LIN {X 0,Y 386.011,Z 375.259,A -85,B 0,C 180,E1 14858.04,E2 14858.04} C_VEL
LIN {X 0,Y 386.531,Z 375.685,A -85,B 0,C 180,E1 14854.451,E2 14854.451} C_VEL
LIN {X 0,Y 386.714,Z 375.838,A -85,B 0,C 180,E1 14850.889,E2 14850.889} C_VEL
LIN {X 0,Y 386.655,Z 375.781,A -85,B 0,C 180,E1 14847.184,E2 14847.184} C_VEL
LIN {X 0,Y 386.291,Z 375.479,A -85,B 0,C 180,E1 14843.61,E2 14843.61} C_VEL
LIN {X 0,Y 385.591,Z 374.785,A -85,B 0,C 180,E1 14839.693,E2 14839.693} C_VEL
LIN {X 0,Y 384.724,Z 373.685,A -85,B 0,C 180,E1 14836.167,E2 14836.167} C_VEL
LIN {X 0,Y 383.625,Z 371.619,A -85,B 0,C 180,E1 14832.559,E2 14832.559} C_VEL
LIN {X 0,Y 382.556,Z 370.431,A -85,B 0,C 180,E1 14829.766,E2 14829.766} C_VEL
LIN {X 0,Y 380.821,Z 369.656,A -85,B 0,C 180,E1 14826.151,E2 14826.151} C_VEL
LIN {X 0,Y 378.919,Z 368.36,A -85,B 0,C 180,E1 14822.669,E2 14822.669} C_VEL
LIN {X 0,Y 377.138,Z 366.192,A -85,B 0,C 180,E1 14819.5,E2 14819.5} C_VEL
LIN {X 0,Y 375.495,Z 363.505,A -85,B 0,C 180,E1 14816.731,E2 14816.731} C_VEL
LIN {X 0,Y 372.832,Z 362.159,A -85,B 0,C 180,E1 14813.051,E2 14813.051} C_VEL
LIN {X 0,Y 370.445,Z 359.93,A -85,B 0,C 180,E1 14809.83,E2 14809.83} C_VEL
LIN {X 0,Y 368.756,Z 357.1,A -85,B 0,C 180,E1 14807.52,E2 14807.52} C_VEL
LIN {X 0,Y 367.813,Z 356.251,A -85,B 0,C 180,E1 14806.31,E2 14806.31} C_VEL
LIN {X 0,Y 364.925,Z 354.532,A -85,B 0,C 180,E1 14802.985,E2 14802.985} C_VEL
LIN {X 0,Y 362.696,Z 352.012,A -85,B 0,C 180,E1 14800.378,E2 14800.378} C_VEL
LIN {X 0,Y 361.179,Z 349.438,A -85,B 0,C 180,E1 14798.526,E2 14798.526} C_VEL
LIN {X 0,Y 358.071,Z 347.716,A -85,B 0,C 180,E1 14795.311,E2 14795.311} C_VEL
LIN {X 0,Y 355.633,Z 344.996,A -85,B 0,C 180,E1 14792.67,E2 14792.67} C_VEL
LIN {X 0,Y 354.249,Z 342.492,A -85,B 0,C 180,E1 14791.099,E2 14791.099} C_VEL
LIN {X 0,Y 350.886,Z 340.633,A -85,B 0,C 180,E1 14787.86,E2 14787.86} C_VEL
LIN {X 0,Y 348.108,Z 337.648,A -85,B 0,C 180,E1 14785.43,E2 14785.43} C_VEL
LIN {X 0,Y 346.58,Z 335.327,A -85,B 0,C 180,E1 14784.183,E2 14784.183} C_VEL
LIN {X 0,Y 344.787,Z 334.431,A -85,B 0,C 180,E1 14782.943,E2 14782.943} C_VEL
LIN {X 0,Y 343.15,Z 334.686,A -85,B 0,C 180,E1 14781.962,E2 14781.962} C_VEL
LIN {X 0,Y 339.462,Z 337.058,A -85,B 0,C 180,E1 14780.04,E2 14780.04} C_VEL
LIN {X 0,Y 337.971,Z 336.456,A -85,B 0,C 180,E1 14779.212,E2 14779.212} C_VEL
LIN {X 0,Y 337.791,Z 336.192,A -85,B 0,C 180,E1 14779.1,E2 14779.1} C_VEL
LIN {X 0,Y 333.793,Z 333.025,A -85,B 0,C 180,E1 14776.712,E2 14776.712} C_VEL
LIN {X 0,Y 331.304,Z 329.103,A -85,B 0,C 180,E1 14774.864,E2 14774.864} C_VEL
LIN {X 0,Y 327.846,Z 326.408,A -85,B 0,C 180,E1 14772.058,E2 14772.058} C_VEL
LIN {X 0,Y 325.939,Z 322.868,A -85,B 0,C 180,E1 14769.892,E2 14769.892} C_VEL
LIN {X 0,Y 321.747,Z 319.853,A -85,B 0,C 180,E1 14761.425,E2 14761.425} C_VEL
LIN {X 0,Y 322.04,Z 320.213,A -85,B 0,C 180,E1 14757.331,E2 14757.331} C_VEL
LIN {X 0,Y 326.157,Z 323.109,A -85,B 0,C 180,E1 14750.293,E2 14750.293} C_VEL
LIN {X 0,Y 327.926,Z 326.507,A -85,B 0,C 180,E1 14748.302,E2 14748.302} C_VEL
LIN {X 0,Y 331.172,Z 329.042,A -85,B 0,C 180,E1 14745.666,E2 14745.666} C_VEL
LIN {X 0,Y 331.836,Z 329.903,A -85,B 0,C 180,E1 14745.16,E2 14745.16} C_VEL
LIN {X 0,Y 334.411,Z 333.737,A -85,B 0,C 180,E1 14743.32,E2 14743.32} C_VEL
LIN {X 0,Y 336.959,Z 335.929,A -85,B 0,C 180,E1 14741.802,E2 14741.802} C_VEL
LIN {X 0,Y 340.182,Z 340.253,A -85,B 0,C 180,E1 14739.976,E2 14739.976} C_VEL
LIN {X 0,Y 341.916,Z 342.055,A -85,B 0,C 180,E1 14739.099,E2 14739.099} C_VEL
LIN {X 0,Y 345.521,Z 346.558,A -85,B 0,C 180,E1 14737.364,E2 14737.364} C_VEL
LIN {X 0,Y 351.232,Z 353.852,A -85,B 0,C 180,E1 14734.903,E2 14734.903} C_VEL
LIN {X 0,Y 355.157,Z 359.117,A -85,B 0,C 180,E1 14733.364,E2 14733.364} C_VEL
LIN {X 0,Y 362.926,Z 371.553,A -85,B 0,C 180,E1 14730.543,E2 14730.543} C_VEL
LIN {X 0,Y 370.435,Z 384.324,A -85,B 0,C 180,E1 14728.106,E2 14728.106} C_VEL
LIN {X 0,Y 378.916,Z 400.148,A -85,B 0,C 180,E1 14725.596,E2 14725.596} C_VEL
LIN {X 0,Y 379.902,Z 402.489,A -85,B 0,C 180,E1 14725.306,E2 14725.306} C_VEL
LIN {X 0,Y 368.607,Z 600.449,A -85,B 0,C 180,E1 14721.342,E2 14721.342} C_VEL
LIN {X 0,Y 366.108,Z 623.413,A -85,B 0,C 180,E1 14720.702,E2 14720.702} C_VEL
LIN {X 0,Y 363.074,Z 642.585,A -85,B 0,C 180,E1 14719.956,E2 14719.956} C_VEL
LIN {X 0,Y 359.795,Z 659.806,A -85,B 0,C 180,E1 14719.1,E2 14719.1} C_VEL
LIN {X 0,Y 355.353,Z 679.953,A -85,B 0,C 180,E1 14717.85,E2 14717.85} C_VEL
LIN {X 0,Y 350.278,Z 699.216,A -85,B 0,C 180,E1 14716.34,E2 14716.34} C_VEL
LIN {X 0,Y 345.77,Z 714.793,A -85,B 0,C 180,E1 14714.874,E2 14714.874} C_VEL
LIN {X 0,Y 340.805,Z 730.632,A -85,B 0,C 180,E1 14713.122,E2 14713.122} C_VEL
LIN {X 0,Y 334.365,Z 749.665,A -85,B 0,C 180,E1 14710.576,E2 14710.576} C_VEL
LIN {X 0,Y 329.444,Z 763.462,A -85,B 0,C 180,E1 14708.363,E2 14708.363} C_VEL
LIN {X 0,Y 324.527,Z 776.993,A -85,B 0,C 180,E1 14705.829,E2 14705.829} C_VEL
LIN {X 0,Y 318.929,Z 792.167,A -85,B 0,C 180,E1 14702.417,E2 14702.417} C_VEL
LIN {X 0,Y 314.992,Z 803.107,A -85,B 0,C 180,E1 14699.472,E2 14699.472} C_VEL
LIN {X 0,Y 311.188,Z 814.397,A -85,B 0,C 180,E1 14695.888,E2 14695.888} C_VEL
LIN {X 0,Y 308.203,Z 824.017,A -85,B 0,C 180,E1 14692.105,E2 14692.105} C_VEL
LIN {X 0,Y 306.371,Z 830.914,A -85,B 0,C 180,E1 14688.839,E2 14688.839} C_VEL
LIN {X 0,Y 305.04,Z 837.21,A -85,B 0,C 180,E1 14685.202,E2 14685.202} C_VEL
LIN {X 0,Y 304.236,Z 842.687,A -85,B 0,C 180,E1 14680.988,E2 14680.988} C_VEL
LIN {X 0,Y 303.996,Z 845.821,A -85,B 0,C 180,E1 14677.56,E2 14677.56} C_VEL
LIN {X 0,Y 303.952,Z 847.721,A -85,B 0,C 180,E1 14674.339,E2 14674.339} C_VEL
LIN {X 0,Y 303.961,Z 848.599,A -85,B 0,C 180,E1 14671.131,E2 14671.131} C_VEL
LIN {X 0,Y 303.955,Z 848.433,A -85,B 0,C 180,E1 14667.738,E2 14667.738} C_VEL
LIN {X 0,Y 303.963,Z 846.79,A -85,B 0,C 180,E1 14663.768,E2 14663.768} C_VEL
LIN {X 0,Y 304.125,Z 843.858,A -85,B 0,C 180,E1 14660.157,E2 14660.157} C_VEL
LIN {X 0,Y 304.586,Z 839.894,A -85,B 0,C 180,E1 14656.716,E2 14656.716} C_VEL
LIN {X 0,Y 305.586,Z 834.412,A -85,B 0,C 180,E1 14653.071,E2 14653.071} C_VEL
LIN {X 0,Y 307.593,Z 826.186,A -85,B 0,C 180,E1 14648.85,E2 14648.85} C_VEL
LIN {X 0,Y 309.881,Z 818.374,A -85,B 0,C 180,E1 14645.607,E2 14645.607} C_VEL
LIN {X 0,Y 312.881,Z 809.224,A -85,B 0,C 180,E1 14642.396,E2 14642.396} C_VEL
LIN {X 0,Y 317.628,Z 795.763,A -85,B 0,C 180,E1 14638.498,E2 14638.498} C_VEL
LIN {X 0,Y 321.804,Z 784.311,A -85,B 0,C 180,E1 14635.738,E2 14635.738} C_VEL
LIN {X 0,Y 326.663,Z 771.157,A -85,B 0,C 180,E1 14633.023,E2 14633.023} C_VEL
LIN {X 0,Y 332.804,Z 754.126,A -85,B 0,C 180,E1 14630.103,E2 14630.103} C_VEL
LIN {X 0,Y 337.815,Z 739.613,A -85,B 0,C 180,E1 14628.018,E2 14628.018} C_VEL
LIN {X 0,Y 343.135,Z 723.386,A -85,B 0,C 180,E1 14626.032,E2 14626.032} C_VEL
LIN {X 0,Y 348.815,Z 704.431,A -85,B 0,C 180,E1 14624.12,E2 14624.12} C_VEL
LIN {X 0,Y 353.278,Z 687.915,A -85,B 0,C 180,E1 14622.741,E2 14622.741} C_VEL
LIN {X 0,Y 357.676,Z 669.757,A -85,B 0,C 180,E1 14621.483,E2 14621.483} C_VEL
LIN {X 0,Y 362.253,Z 647.281,A -85,B 0,C 180,E1 14620.257,E2 14620.257} C_VEL
LIN {X 0,Y 365.247,Z 629.114,A -85,B 0,C 180,E1 14619.502,E2 14619.502} C_VEL
LIN {X 0,Y 367.731,Z 609.909,A -85,B 0,C 180,E1 14618.895,E2 14618.895} C_VEL
LIN {X 0,Y 369.86,Z 580.866,A -85,B 0,C 180,E1 14618.239,E2 14618.239} C_VEL
LIN {X 0,Y 379.865,Z 402.063,A -85,B 0,C 180,E1 14614.672,E2 14614.672} C_VEL
LIN {X 0,Y 372.117,Z 387.455,A -85,B 0,C 180,E1 14612.415,E2 14612.415} C_VEL
LIN {X 0,Y 365.916,Z 376.518,A -85,B 0,C 180,E1 14610.456,E2 14610.456} C_VEL
LIN {X 0,Y 360.022,Z 366.838,A -85,B 0,C 180,E1 14608.443,E2 14608.443} C_VEL
LIN {X 0,Y 353.711,Z 357.015,A -85,B 0,C 180,E1 14606.076,E2 14606.076} C_VEL
LIN {X 0,Y 349.294,Z 351.398,A -85,B 0,C 180,E1 14604.298,E2 14604.298} C_VEL
LIN {X 0,Y 345.346,Z 346.397,A -85,B 0,C 180,E1 14602.558,E2 14602.558} C_VEL
LIN {X 0,Y 341.766,Z 341.796,A -85,B 0,C 180,E1 14600.821,E2 14600.821} C_VEL
LIN {X 0,Y 337.557,Z 336.961,A -85,B 0,C 180,E1 14598.567,E2 14598.567} C_VEL
LIN {X 0,Y 336.628,Z 335.401,A -85,B 0,C 180,E1 14597.993,E2 14597.993} C_VEL
LIN {X 0,Y 333.408,Z 332.568,A -85,B 0,C 180,E1 14596.016,E2 14596.016} C_VEL
LIN {X 0,Y 331.41,Z 329.161,A -85,B 0,C 180,E1 14594.502,E2 14594.502} C_VEL
LIN {X 0,Y 327.926,Z 326.505,A -85,B 0,C 180,E1 14591.698,E2 14591.698} C_VEL
LIN {X 0,Y 326.003,Z 322.973,A -85,B 0,C 180,E1 14589.533,E2 14589.533} C_VEL
LIN {X 0,Y 321.774,Z 319.91,A -85,B 0,C 180,E1 14581.246,E2 14581.246} C_VEL
LIN {X 0,Y 321.978,Z 320.151,A -85,B 0,C 180,E1 14577.152,E2 14577.152} C_VEL
LIN {X 0,Y 326.163,Z 323.134,A -85,B 0,C 180,E1 14569.848,E2 14569.848} C_VEL
LIN {X 0,Y 328.026,Z 326.626,A -85,B 0,C 180,E1 14567.77,E2 14567.77} C_VEL
LIN {X 0,Y 331.694,Z 329.582,A -85,B 0,C 180,E1 14564.841,E2 14564.841} C_VEL
LIN {X 0,Y 334.299,Z 333.596,A -85,B 0,C 180,E1 14562.956,E2 14562.956} C_VEL
LIN {X 0,Y 337.907,Z 336.386,A -85,B 0,C 180,E1 14560.826,E2 14560.826} C_VEL
LIN {X 0,Y 340.872,Z 340.262,A -85,B 0,C 180,E1 14558.942,E2 14558.942} C_VEL
LIN {X 0,Y 344.246,Z 342.664,A -85,B 0,C 180,E1 14556.733,E2 14556.733} C_VEL
LIN {X 0,Y 345.62,Z 343.626,A -85,B 0,C 180,E1 14555.745,E2 14555.745} C_VEL
LIN {X 0,Y 347.956,Z 346.835,A -85,B 0,C 180,E1 14553.827,E2 14553.827} C_VEL
LIN {X 0,Y 350.713,Z 349.153,A -85,B 0,C 180,E1 14551.383,E2 14551.383} C_VEL
LIN {X 0,Y 353.32,Z 350.716,A -85,B 0,C 180,E1 14548.811,E2 14548.811} C_VEL
LIN {X 0,Y 355.344,Z 354.06,A -85,B 0,C 180,E1 14546.53,E2 14546.53} C_VEL
LIN {X 0,Y 358.406,Z 356.549,A -85,B 0,C 180,E1 14543.345,E2 14543.345} C_VEL
LIN {X 0,Y 360.372,Z 357.729,A -85,B 0,C 180,E1 14541.27,E2 14541.27} C_VEL
LIN {X 0,Y 362.586,Z 361.266,A -85,B 0,C 180,E1 14538.562,E2 14538.562} C_VEL
LIN {X 0,Y 365.41,Z 363.514,A -85,B 0,C 180,E1 14535.314,E2 14535.314} C_VEL
LIN {X 0,Y 367.493,Z 364.663,A -85,B 0,C 180,E1 14532.857,E2 14532.857} C_VEL
LIN {X 0,Y 369.237,Z 367.669,A -85,B 0,C 180,E1 14530.455,E2 14530.455} C_VEL
LIN {X 0,Y 371.484,Z 369.86,A -85,B 0,C 180,E1 14527.439,E2 14527.439} C_VEL
LIN {X 0,Y 374.035,Z 371.221,A -85,B 0,C 180,E1 14523.964,E2 14523.964} C_VEL
LIN {X 0,Y 375.036,Z 372.228,A -85,B 0,C 180,E1 14522.402,E2 14522.402} C_VEL
LIN {X 0,Y 376.884,Z 375.227,A -85,B 0,C 180,E1 14519.212,E2 14519.212} C_VEL
LIN {X 0,Y 378.863,Z 377.028,A -85,B 0,C 180,E1 14515.645,E2 14515.645} C_VEL
LIN {X 0,Y 380.652,Z 377.988,A -85,B 0,C 180,E1 14512.224,E2 14512.224} C_VEL
LIN {X 0,Y 382.225,Z 378.874,A -85,B 0,C 180,E1 14508.747,E2 14508.747} C_VEL
LIN {X 0,Y 383.348,Z 380.95,A -85,B 0,C 180,E1 14505.195,E2 14505.195} C_VEL
LIN {X 0,Y 384.312,Z 382.396,A -85,B 0,C 180,E1 14501.708,E2 14501.708} C_VEL
LIN {X 0,Y 385.001,Z 383.161,A -85,B 0,C 180,E1 14498.212,E2 14498.212} C_VEL
LIN {X 0,Y 385.54,Z 383.608,A -85,B 0,C 180,E1 14494.611,E2 14494.611} C_VEL
LIN {X 0,Y 385.734,Z 383.773,A -85,B 0,C 180,E1 14491.04,E2 14491.04} C_VEL
LIN {X 0,Y 385.691,Z 383.733,A -85,B 0,C 180,E1 14487.326,E2 14487.326} C_VEL
LIN {X 0,Y 385.333,Z 383.446,A -85,B 0,C 180,E1 14483.744,E2 14483.744} C_VEL
LIN {X 0,Y 384.675,Z 382.815,A -85,B 0,C 180,E1 14479.971,E2 14479.971} C_VEL
LIN {X 0,Y 383.829,Z 381.752,A -85,B 0,C 180,E1 14476.441,E2 14476.441} C_VEL
LIN {X 0,Y 382.796,Z 379.785,A -85,B 0,C 180,E1 14472.937,E2 14472.937} C_VEL
LIN {X 0,Y 381.65,Z 378.409,A -85,B 0,C 180,E1 14469.929,E2 14469.929} C_VEL
LIN {X 0,Y 379.891,Z 377.628,A -85,B 0,C 180,E1 14466.254,E2 14466.254} C_VEL
LIN {X 0,Y 377.969,Z 376.351,A -85,B 0,C 180,E1 14462.727,E2 14462.727} C_VEL
LIN {X 0,Y 376.128,Z 374.16,A -85,B 0,C 180,E1 14459.461,E2 14459.461} C_VEL
LIN {X 0,Y 374.453,Z 371.411,A -85,B 0,C 180,E1 14456.63,E2 14456.63} C_VEL
LIN {X 0,Y 371.78,Z 370.066,A -85,B 0,C 180,E1 14452.958,E2 14452.958} C_VEL
LIN {X 0,Y 369.397,Z 367.862,A -85,B 0,C 180,E1 14449.756,E2 14449.756} C_VEL
LIN {X 0,Y 367.651,Z 365.01,A -85,B 0,C 180,E1 14447.378,E2 14447.378} C_VEL
LIN {X 0,Y 366.773,Z 364.175,A -85,B 0,C 180,E1 14446.254,E2 14446.254} C_VEL
LIN {X 0,Y 363.902,Z 362.485,A -85,B 0,C 180,E1 14442.953,E2 14442.953} C_VEL
LIN {X 0,Y 361.585,Z 359.928,A -85,B 0,C 180,E1 14440.255,E2 14440.255} C_VEL
LIN {X 0,Y 359.927,Z 357.29,A -85,B 0,C 180,E1 14438.278,E2 14438.278} C_VEL
LIN {X 0,Y 356.842,Z 355.495,A -85,B 0,C 180,E1 14435.058,E2 14435.058} C_VEL
LIN {X 0,Y 354.391,Z 352.74,A -85,B 0,C 180,E1 14432.415,E2 14432.415} C_VEL
LIN {X 0,Y 353.016,Z 350.332,A -85,B 0,C 180,E1 14430.841,E2 14430.841} C_VEL
LIN {X 0,Y 349.525,Z 348.336,A -85,B 0,C 180,E1 14427.53,E2 14427.53} C_VEL
LIN {X 0,Y 346.676,Z 345.239,A -85,B 0,C 180,E1 14425.085,E2 14425.085} C_VEL
LIN {X 0,Y 345.201,Z 343.121,A -85,B 0,C 180,E1 14423.923,E2 14423.923} C_VEL
LIN {X 0,Y 341.517,Z 340.835,A -85,B 0,C 180,E1 14421.467,E2 14421.467} C_VEL
LIN {X 0,Y 338.685,Z 337.568,A -85,B 0,C 180,E1 14419.658,E2 14419.658} C_VEL
LIN {X 0,Y 337.791,Z 336.192,A -85,B 0,C 180,E1 14419.1,E2 14419.1} C_VEL
LIN {X 0,Y 336.204,Z 334.673,A -85,B 0,C 180,E1 14418.145,E2 14418.145} C_VEL
LIN {X 0,Y 333.608,Z 334.681,A -85,B 0,C 180,E1 14416.692,E2 14416.692} C_VEL
LIN {X 0,Y 329.248,Z 336.176,A -85,B 0,C 180,E1 14414.065,E2 14414.065} C_VEL
LIN {X 0,Y 328.115,Z 335.75,A -85,B 0,C 180,E1 14413.204,E2 14413.204} C_VEL
LIN {X 0,Y 325.562,Z 332.515,A -85,B 0,C 180,E1 14410.708,E2 14410.708} C_VEL
LIN {X 0,Y 324.672,Z 330.612,A -85,B 0,C 180,E1 14409.573,E2 14409.573} C_VEL
LIN {X 0,Y 320.755,Z 327.77,A -85,B 0,C 180,E1 14401.25,E2 14401.25} C_VEL
LIN {X 0,Y 321.109,Z 328.228,A -85,B 0,C 180,E1 14397.144,E2 14397.144} C_VEL
LIN {X 0,Y 324.884,Z 330.824,A -85,B 0,C 180,E1 14390.612,E2 14390.612} C_VEL
LIN {X 0,Y 326.681,Z 334.309,A -85,B 0,C 180,E1 14388.525,E2 14388.525} C_VEL
LIN {X 0,Y 330.243,Z 337.376,A -85,B 0,C 180,E1 14385.58,E2 14385.58} C_VEL
LIN {X 0,Y 332.929,Z 341.425,A -85,B 0,C 180,E1 14383.602,E2 14383.602} C_VEL
LIN {X 0,Y 335.288,Z 343.541,A -85,B 0,C 180,E1 14382.157,E2 14382.157} C_VEL
LIN {X 0,Y 338.76,Z 348.09,A -85,B 0,C 180,E1 14380.158,E2 14380.158} C_VEL
LIN {X 0,Y 340.22,Z 349.818,A -85,B 0,C 180,E1 14379.395,E2 14379.395} C_VEL
LIN {X 0,Y 344.789,Z 355.602,A -85,B 0,C 180,E1 14377.178,E2 14377.178} C_VEL
LIN {X 0,Y 349.224,Z 361.396,A -85,B 0,C 180,E1 14375.246,E2 14375.246} C_VEL
LIN {X 0,Y 352.608,Z 366.012,A -85,B 0,C 180,E1 14373.882,E2 14373.882} C_VEL
LIN {X 0,Y 359.912,Z 377.94,A -85,B 0,C 180,E1 14371.139,E2 14371.139} C_VEL
LIN {X 0,Y 367.152,Z 390.522,A -85,B 0,C 180,E1 14368.704,E2 14368.704} C_VEL
LIN {X 0,Y 375.167,Z 405.842,A -85,B 0,C 180,E1 14366.243,E2 14366.243} C_VEL
LIN {X 0,Y 363.634,Z 600.313,A -85,B 0,C 180,E1 14362.328,E2 14362.328} C_VEL
LIN {X 0,Y 361.018,Z 623.485,A -85,B 0,C 180,E1 14361.678,E2 14361.678} C_VEL
LIN {X 0,Y 357.939,Z 642.334,A -85,B 0,C 180,E1 14360.945,E2 14360.945} C_VEL
LIN {X 0,Y 354.408,Z 660.251,A -85,B 0,C 180,E1 14360.05,E2 14360.05} C_VEL
LIN {X 0,Y 349.693,Z 680.754,A -85,B 0,C 180,E1 14358.76,E2 14358.76} C_VEL
LIN {X 0,Y 344.476,Z 699.746,A -85,B 0,C 180,E1 14357.25,E2 14357.25} C_VEL
LIN {X 0,Y 339.882,Z 715.011,A -85,B 0,C 180,E1 14355.797,E2 14355.797} C_VEL
LIN {X 0,Y 334.325,Z 732.04,A -85,B 0,C 180,E1 14353.884,E2 14353.884} C_VEL
LIN {X 0,Y 327.936,Z 749.995,A -85,B 0,C 180,E1 14351.422,E2 14351.422} C_VEL
LIN {X 0,Y 322.817,Z 763.703,A -85,B 0,C 180,E1 14349.185,E2 14349.185} C_VEL
LIN {X 0,Y 317.192,Z 778.525,A -85,B 0,C 180,E1 14346.342,E2 14346.342} C_VEL
LIN {X 0,Y 311.676,Z 792.629,A -85,B 0,C 180,E1 14343.048,E2 14343.048} C_VEL
LIN {X 0,Y 307.56,Z 803.491,A -85,B 0,C 180,E1 14340.042,E2 14340.042} C_VEL
LIN {X 0,Y 303.404,Z 815.121,A -85,B 0,C 180,E1 14336.205,E2 14336.205} C_VEL
LIN {X 0,Y 300.428,Z 824.194,A -85,B 0,C 180,E1 14332.502,E2 14332.502} C_VEL
LIN {X 0,Y 298.501,Z 831.011,A -85,B 0,C 180,E1 14329.163,E2 14329.163} C_VEL
LIN {X 0,Y 296.983,Z 837.869,A -85,B 0,C 180,E1 14325.024,E2 14325.024} C_VEL
LIN {X 0,Y 296.223,Z 842.826,A -85,B 0,C 180,E1 14320.895,E2 14320.895} C_VEL
LIN {X 0,Y 295.998,Z 845.709,A -85,B 0,C 180,E1 14317.57,E2 14317.57} C_VEL
LIN {X 0,Y 295.954,Z 847.555,A -85,B 0,C 180,E1 14314.262,E2 14314.262} C_VEL
LIN {X 0,Y 295.962,Z 848.406,A -85,B 0,C 180,E1 14310.774,E2 14310.774} C_VEL
LIN {X 0,Y 295.953,Z 847.969,A -85,B 0,C 180,E1 14306.708,E2 14306.708} C_VEL
LIN {X 0,Y 295.992,Z 845.987,A -85,B 0,C 180,E1 14302.82,E2 14302.82} C_VEL
LIN {X 0,Y 296.18,Z 843.216,A -85,B 0,C 180,E1 14299.497,E2 14299.497} C_VEL
LIN {X 0,Y 296.737,Z 839.135,A -85,B 0,C 180,E1 14295.96,E2 14295.96} C_VEL
LIN {X 0,Y 298.065,Z 832.867,A -85,B 0,C 180,E1 14291.823,E2 14291.823} C_VEL
LIN {X 0,Y 300.166,Z 825.062,A -85,B 0,C 180,E1 14287.89,E2 14287.89} C_VEL
LIN {X 0,Y 302.693,Z 817.119,A -85,B 0,C 180,E1 14284.57,E2 14284.57} C_VEL
LIN {X 0,Y 306.647,Z 806.055,A -85,B 0,C 180,E1 14280.72,E2 14280.72} C_VEL
LIN {X 0,Y 311.124,Z 794.067,A -85,B 0,C 180,E1 14277.324,E2 14277.324} C_VEL
LIN {X 0,Y 315.678,Z 782.29,A -85,B 0,C 180,E1 14274.489,E2 14274.489} C_VEL
LIN {X 0,Y 321.72,Z 766.69,A -85,B 0,C 180,E1 14271.343,E2 14271.343} C_VEL
LIN {X 0,Y 327.117,Z 752.209,A -85,B 0,C 180,E1 14268.917,E2 14268.917} C_VEL
LIN {X 0,Y 332.336,Z 737.697,A -85,B 0,C 180,E1 14266.845,E2 14266.845} C_VEL
LIN {X 0,Y 338.829,Z 718.396,A -85,B 0,C 180,E1 14264.551,E2 14264.551} C_VEL
LIN {X 0,Y 343.97,Z 701.484,A -85,B 0,C 180,E1 14262.904,E2 14262.904} C_VEL
LIN {X 0,Y 348.617,Z 684.702,A -85,B 0,C 180,E1 14261.536,E2 14261.536} C_VEL
LIN {X 0,Y 353.809,Z 663.186,A -85,B 0,C 180,E1 14260.115,E2 14260.115} C_VEL
LIN {X 0,Y 357.516,Z 644.683,A -85,B 0,C 180,E1 14259.163,E2 14259.163} C_VEL
LIN {X 0,Y 360.462,Z 627.071,A -85,B 0,C 180,E1 14258.45,E2 14258.45} C_VEL
LIN {X 0,Y 363.272,Z 604.983,A -85,B 0,C 180,E1 14257.779,E2 14257.779} C_VEL
LIN {X 0,Y 365.865,Z 564.336,A -85,B 0,C 180,E1 14256.921,E2 14256.921} C_VEL
LIN {X 0,Y 375.12,Z 405.682,A -85,B 0,C 180,E1 14253.741,E2 14253.741} C_VEL
LIN {X 0,Y 366.931,Z 390.135,A -85,B 0,C 180,E1 14251.226,E2 14251.226} C_VEL
LIN {X 0,Y 358.498,Z 375.402,A -85,B 0,C 180,E1 14248.348,E2 14248.348} C_VEL
LIN {X 0,Y 351.191,Z 363.936,A -85,B 0,C 180,E1 14245.552,E2 14245.552} C_VEL
LIN {X 0,Y 346.872,Z 358.349,A -85,B 0,C 180,E1 14243.755,E2 14243.755} C_VEL
LIN {X 0,Y 343.357,Z 353.771,A -85,B 0,C 180,E1 14242.154,E2 14242.154} C_VEL
LIN {X 0,Y 339.072,Z 348.368,A -85,B 0,C 180,E1 14240.002,E2 14240.002} C_VEL
LIN {X 0,Y 335.547,Z 343.994,A -85,B 0,C 180,E1 14238.008,E2 14238.008} C_VEL
LIN {X 0,Y 334.538,Z 342.755,A -85,B 0,C 180,E1 14237.39,E2 14237.39} C_VEL
LIN {X 0,Y 331.479,Z 339.607,A -85,B 0,C 180,E1 14235.393,E2 14235.393} C_VEL
LIN {X 0,Y 329.983,Z 336.925,A -85,B 0,C 180,E1 14234.207,E2 14234.207} C_VEL
LIN {X 0,Y 326.593,Z 334.198,A -85,B 0,C 180,E1 14231.389,E2 14231.389} C_VEL
LIN {X 0,Y 324.731,Z 330.717,A -85,B 0,C 180,E1 14229.213,E2 14229.213} C_VEL
LIN {X 0,Y 320.762,Z 327.785,A -85,B 0,C 180,E1 14220.893,E2 14220.893} C_VEL
LIN {X 0,Y 321.09,Z 328.196,A -85,B 0,C 180,E1 14216.787,E2 14216.787} C_VEL
LIN {X 0,Y 324.957,Z 330.992,A -85,B 0,C 180,E1 14210.078,E2 14210.078} C_VEL
LIN {X 0,Y 326.78,Z 334.428,A -85,B 0,C 180,E1 14207.991,E2 14207.991} C_VEL
LIN {X 0,Y 330.207,Z 337.286,A -85,B 0,C 180,E1 14205.175,E2 14205.175} C_VEL
LIN {X 0,Y 332.949,Z 341.421,A -85,B 0,C 180,E1 14203.154,E2 14203.154} C_VEL
LIN {X 0,Y 336.392,Z 344.171,A -85,B 0,C 180,E1 14201.096,E2 14201.096} C_VEL
LIN {X 0,Y 339.393,Z 347.964,A -85,B 0,C 180,E1 14199.207,E2 14199.207} C_VEL
LIN {X 0,Y 343.073,Z 350.556,A -85,B 0,C 180,E1 14196.831,E2 14196.831} C_VEL
LIN {X 0,Y 344.243,Z 351.389,A -85,B 0,C 180,E1 14196.007,E2 14196.007} C_VEL
LIN {X 0,Y 346.724,Z 354.671,A -85,B 0,C 180,E1 14194.003,E2 14194.003} C_VEL
LIN {X 0,Y 349.424,Z 356.947,A -85,B 0,C 180,E1 14191.641,E2 14191.641} C_VEL
LIN {X 0,Y 352.158,Z 358.611,A -85,B 0,C 180,E1 14188.991,E2 14188.991} C_VEL
LIN {X 0,Y 354.277,Z 361.998,A -85,B 0,C 180,E1 14186.61,E2 14186.61} C_VEL
LIN {X 0,Y 357.344,Z 364.465,A -85,B 0,C 180,E1 14183.418,E2 14183.418} C_VEL
LIN {X 0,Y 359.21,Z 365.622,A -85,B 0,C 180,E1 14181.428,E2 14181.428} C_VEL
LIN {X 0,Y 361.542,Z 369.207,A -85,B 0,C 180,E1 14178.627,E2 14178.627} C_VEL
LIN {X 0,Y 364.451,Z 371.48,A -85,B 0,C 180,E1 14175.279,E2 14175.279} C_VEL
LIN {X 0,Y 366.394,Z 372.568,A -85,B 0,C 180,E1 14173.001,E2 14173.001} C_VEL
LIN {X 0,Y 368.244,Z 375.668,A -85,B 0,C 180,E1 14170.46,E2 14170.46} C_VEL
LIN {X 0,Y 370.538,Z 377.847,A -85,B 0,C 180,E1 14167.382,E2 14167.382} C_VEL
LIN {X 0,Y 373.157,Z 379.196,A -85,B 0,C 180,E1 14163.836,E2 14163.836} C_VEL
LIN {X 0,Y 373.979,Z 380.168,A -85,B 0,C 180,E1 14162.505,E2 14162.505} C_VEL
LIN {X 0,Y 375.882,Z 383.172,A -85,B 0,C 180,E1 14159.251,E2 14159.251} C_VEL
LIN {X 0,Y 377.848,Z 384.949,A -85,B 0,C 180,E1 14155.719,E2 14155.719} C_VEL
LIN {X 0,Y 379.636,Z 385.917,A -85,B 0,C 180,E1 14152.287,E2 14152.287} C_VEL
LIN {X 0,Y 381.238,Z 386.811,A -85,B 0,C 180,E1 14148.777,E2 14148.777} C_VEL
LIN {X 0,Y 382.358,Z 388.892,A -85,B 0,C 180,E1 14145.22,E2 14145.22} C_VEL
LIN {X 0,Y 383.329,Z 390.334,A -85,B 0,C 180,E1 14141.739,E2 14141.739} C_VEL
LIN {X 0,Y 384.019,Z 391.1,A -85,B 0,C 180,E1 14138.233,E2 14138.233} C_VEL
LIN {X 0,Y 384.566,Z 391.548,A -85,B 0,C 180,E1 14134.623,E2 14134.623} C_VEL
LIN {X 0,Y 384.757,Z 391.713,A -85,B 0,C 180,E1 14131.042,E2 14131.042} C_VEL
LIN {X 0,Y 384.729,Z 391.685,A -85,B 0,C 180,E1 14127.468,E2 14127.468} C_VEL
LIN {X 0,Y 384.366,Z 391.414,A -85,B 0,C 180,E1 14123.878,E2 14123.878} C_VEL
LIN {X 0,Y 383.769,Z 390.838,A -85,B 0,C 180,E1 14120.25,E2 14120.25} C_VEL
LIN {X 0,Y 382.912,Z 389.786,A -85,B 0,C 180,E1 14116.716,E2 14116.716} C_VEL
LIN {X 0,Y 381.882,Z 387.892,A -85,B 0,C 180,E1 14113.105,E2 14113.105} C_VEL
LIN {X 0,Y 380.793,Z 386.464,A -85,B 0,C 180,E1 14110.202,E2 14110.202} C_VEL
LIN {X 0,Y 379.042,Z 385.649,A -85,B 0,C 180,E1 14106.528,E2 14106.528} C_VEL
LIN {X 0,Y 377.063,Z 384.382,A -85,B 0,C 180,E1 14102.866,E2 14102.866} C_VEL
LIN {X 0,Y 375.21,Z 382.265,A -85,B 0,C 180,E1 14099.583,E2 14099.583} C_VEL
LIN {X 0,Y 373.409,Z 379.317,A -85,B 0,C 180,E1 14096.525,E2 14096.525} C_VEL
LIN {X 0,Y 370.695,Z 377.956,A -85,B 0,C 180,E1 14092.831,E2 14092.831} C_VEL
LIN {X 0,Y 368.368,Z 375.814,A -85,B 0,C 180,E1 14089.704,E2 14089.704} C_VEL
LIN {X 0,Y 366.529,Z 372.881,A -85,B 0,C 180,E1 14087.206,E2 14087.206} C_VEL
LIN {X 0,Y 365.734,Z 372.099,A -85,B 0,C 180,E1 14086.198,E2 14086.198} C_VEL
LIN {X 0,Y 362.825,Z 370.392,A -85,B 0,C 180,E1 14082.861,E2 14082.861} C_VEL
LIN {X 0,Y 360.495,Z 367.872,A -85,B 0,C 180,E1 14080.155,E2 14080.155} C_VEL
LIN {X 0,Y 358.864,Z 365.208,A -85,B 0,C 180,E1 14078.209,E2 14078.209} C_VEL
LIN {X 0,Y 355.774,Z 363.419,A -85,B 0,C 180,E1 14074.982,E2 14074.982} C_VEL
LIN {X 0,Y 353.222,Z 360.599,A -85,B 0,C 180,E1 14072.238,E2 14072.238} C_VEL
LIN {X 0,Y 351.759,Z 358.178,A -85,B 0,C 180,E1 14070.584,E2 14070.584} C_VEL
LIN {X 0,Y 348.496,Z 356.311,A -85,B 0,C 180,E1 14067.511,E2 14067.511} C_VEL
LIN {X 0,Y 345.505,Z 353.252,A -85,B 0,C 180,E1 14064.993,E2 14064.993} C_VEL
LIN {X 0,Y 343.794,Z 350.893,A -85,B 0,C 180,E1 14063.639,E2 14063.639} C_VEL
LIN {X 0,Y 340.057,Z 348.544,A -85,B 0,C 180,E1 14061.202,E2 14061.202} C_VEL
LIN {X 0,Y 337.042,Z 345.145,A -85,B 0,C 180,E1 14059.316,E2 14059.316} C_VEL
LIN {X 0,Y 335.859,Z 343.52,A -85,B 0,C 180,E1 14058.575,E2 14058.575} C_VEL
LIN {X 0,Y 332.325,Z 340.72,A -85,B 0,C 180,E1 14056.428,E2 14056.428} C_VEL
LIN {X 0,Y 329.881,Z 336.873,A -85,B 0,C 180,E1 14054.57,E2 14054.57} C_VEL
LIN {X 0,Y 328.115,Z 335.75,A -85,B 0,C 180,E1 14053.204,E2 14053.204} C_VEL
LIN {X 0,Y 326.283,Z 335.286,A -85,B 0,C 180,E1 14051.676,E2 14051.676} C_VEL
LIN {X 0,Y 322.141,Z 337.687,A -85,B 0,C 180,E1 14047.58,E2 14047.58} C_VEL
LIN {X 0,Y 321.736,Z 337.606,A -85,B 0,C 180,E1 14046.983,E2 14046.983} C_VEL
LIN {X 0,Y 319.766,Z 335.7,A -85,B 0,C 180,E1 14041.075,E2 14041.075} C_VEL
LIN {X 0,Y 320.181,Z 336.251,A -85,B 0,C 180,E1 14036.957,E2 14036.957} C_VEL
LIN {X 0,Y 323.679,Z 338.728,A -85,B 0,C 180,E1 14030.846,E2 14030.846} C_VEL
LIN {X 0,Y 325.527,Z 342.216,A -85,B 0,C 180,E1 14028.663,E2 14028.663} C_VEL
LIN {X 0,Y 328.817,Z 345.161,A -85,B 0,C 180,E1 14025.876,E2 14025.876} C_VEL
LIN {X 0,Y 331.582,Z 349.241,A -85,B 0,C 180,E1 14023.804,E2 14023.804} C_VEL
LIN {X 0,Y 333.695,Z 351.251,A -85,B 0,C 180,E1 14022.475,E2 14022.475} C_VEL
LIN {X 0,Y 337.19,Z 355.78,A -85,B 0,C 180,E1 14020.423,E2 14020.423} C_VEL
LIN {X 0,Y 339.37,Z 358.768,A -85,B 0,C 180,E1 14019.251,E2 14019.251} C_VEL
LIN {X 0,Y 342.87,Z 363.117,A -85,B 0,C 180,E1 14017.542,E2 14017.542} C_VEL
LIN {X 0,Y 347.23,Z 368.923,A -85,B 0,C 180,E1 14015.593,E2 14015.593} C_VEL
LIN {X 0,Y 350.089,Z 372.904,A -85,B 0,C 180,E1 14014.407,E2 14014.407} C_VEL
LIN {X 0,Y 357.036,Z 384.51,A -85,B 0,C 180,E1 14011.707,E2 14011.707} C_VEL
LIN {X 0,Y 364.017,Z 396.912,A -85,B 0,C 180,E1 14009.277,E2 14009.277} C_VEL
LIN {X 0,Y 370.506,Z 409.642,A -85,B 0,C 180,E1 14007.195,E2 14007.195} C_VEL
LIN {X 0,Y 358.781,Z 600.076,A -85,B 0,C 180,E1 14003.344,E2 14003.344} C_VEL
LIN {X 0,Y 356.067,Z 623.355,A -85,B 0,C 180,E1 14002.689,E2 14002.689} C_VEL
LIN {X 0,Y 352.913,Z 642.084,A -85,B 0,C 180,E1 14001.961,E2 14001.961} C_VEL
LIN {X 0,Y 349.276,Z 659.972,A -85,B 0,C 180,E1 14001.068,E2 14001.068} C_VEL
LIN {X 0,Y 344.398,Z 680.502,A -85,B 0,C 180,E1 13999.776,E2 13999.776} C_VEL
LIN {X 0,Y 339,Z 699.493,A -85,B 0,C 180,E1 13998.261,E2 13998.261} C_VEL
LIN {X 0,Y 333.979,Z 715.552,A -85,B 0,C 180,E1 13996.719,E2 13996.719} C_VEL
LIN {X 0,Y 327.867,Z 733.545,A -85,B 0,C 180,E1 13994.661,E2 13994.661} C_VEL
LIN {X 0,Y 321.428,Z 750.723,A -85,B 0,C 180,E1 13992.24,E2 13992.24} C_VEL
LIN {X 0,Y 315.946,Z 764.763,A -85,B 0,C 180,E1 13989.895,E2 13989.895} C_VEL
LIN {X 0,Y 309.525,Z 780.745,A -85,B 0,C 180,E1 13986.697,E2 13986.697} C_VEL
LIN {X 0,Y 304.464,Z 793.09,A -85,B 0,C 180,E1 13983.709,E2 13983.709} C_VEL
LIN {X 0,Y 300.16,Z 803.874,A -85,B 0,C 180,E1 13980.64,E2 13980.64} C_VEL
LIN {X 0,Y 295.606,Z 815.863,A -85,B 0,C 180,E1 13976.517,E2 13976.517} C_VEL
LIN {X 0,Y 292.667,Z 824.372,A -85,B 0,C 180,E1 13972.921,E2 13972.921} C_VEL
LIN {X 0,Y 290.447,Z 831.869,A -85,B 0,C 180,E1 13969.088,E2 13969.088} C_VEL
LIN {X 0,Y 288.87,Z 838.629,A -85,B 0,C 180,E1 13964.635,E2 13964.635} C_VEL
LIN {X 0,Y 288.229,Z 842.793,A -85,B 0,C 180,E1 13960.974,E2 13960.974} C_VEL
LIN {X 0,Y 287.996,Z 845.736,A -85,B 0,C 180,E1 13957.38,E2 13957.38} C_VEL
LIN {X 0,Y 287.954,Z 847.637,A -85,B 0,C 180,E1 13953.583,E2 13953.583} C_VEL
LIN {X 0,Y 287.967,Z 848.184,A -85,B 0,C 180,E1 13949.403,E2 13949.403} C_VEL
LIN {X 0,Y 287.955,Z 847.389,A -85,B 0,C 180,E1 13945.819,E2 13945.819} C_VEL
LIN {X 0,Y 287.999,Z 845.597,A -85,B 0,C 180,E1 13942.419,E2 13942.419} C_VEL
LIN {X 0,Y 288.233,Z 842.769,A -85,B 0,C 180,E1 13939.001,E2 13939.001} C_VEL
LIN {X 0,Y 288.923,Z 838.376,A -85,B 0,C 180,E1 13935.162,E2 13935.162} C_VEL
LIN {X 0,Y 290.54,Z 831.498,A -85,B 0,C 180,E1 13930.709,E2 13930.709} C_VEL
LIN {X 0,Y 292.667,Z 824.372,A -85,B 0,C 180,E1 13927.079,E2 13927.079} C_VEL
LIN {X 0,Y 295.605,Z 815.863,A -85,B 0,C 180,E1 13923.483,E2 13923.483} C_VEL
LIN {X 0,Y 300.16,Z 803.874,A -85,B 0,C 180,E1 13919.36,E2 13919.36} C_VEL
LIN {X 0,Y 304.464,Z 793.09,A -85,B 0,C 180,E1 13916.291,E2 13916.291} C_VEL
LIN {X 0,Y 309.76,Z 780.2,A -85,B 0,C 180,E1 13913.178,E2 13913.178} C_VEL
LIN {X 0,Y 316.071,Z 764.442,A -85,B 0,C 180,E1 13910.048,E2 13910.048} C_VEL
LIN {X 0,Y 321.429,Z 750.721,A -85,B 0,C 180,E1 13907.76,E2 13907.76} C_VEL
LIN {X 0,Y 327.867,Z 733.545,A -85,B 0,C 180,E1 13905.339,E2 13905.339} C_VEL
LIN {X 0,Y 333.979,Z 715.552,A -85,B 0,C 180,E1 13903.281,E2 13903.281} C_VEL
LIN {X 0,Y 339,Z 699.493,A -85,B 0,C 180,E1 13901.739,E2 13901.739} C_VEL
LIN {X 0,Y 344.398,Z 680.502,A -85,B 0,C 180,E1 13900.224,E2 13900.224} C_VEL
LIN {X 0,Y 349.277,Z 659.967,A -85,B 0,C 180,E1 13898.931,E2 13898.931} C_VEL
LIN {X 0,Y 352.914,Z 642.084,A -85,B 0,C 180,E1 13898.039,E2 13898.039} C_VEL
LIN {X 0,Y 356.455,Z 620.89,A -85,B 0,C 180,E1 13897.223,E2 13897.223} C_VEL
LIN {X 0,Y 358.876,Z 598.831,A -85,B 0,C 180,E1 13896.628,E2 13896.628} C_VEL
LIN {X 0,Y 370.515,Z 409.501,A -85,B 0,C 180,E1 13892.802,E2 13892.802} C_VEL
LIN {X 0,Y 362.003,Z 393.102,A -85,B 0,C 180,E1 13890.041,E2 13890.041} C_VEL
LIN {X 0,Y 354.556,Z 380.29,A -85,B 0,C 180,E1 13887.365,E2 13887.365} C_VEL
LIN {X 0,Y 348.795,Z 370.965,A -85,B 0,C 180,E1 13885.058,E2 13885.058} C_VEL
LIN {X 0,Y 344.483,Z 365.291,A -85,B 0,C 180,E1 13883.204,E2 13883.204} C_VEL
LIN {X 0,Y 341.218,Z 360.971,A -85,B 0,C 180,E1 13881.667,E2 13881.667} C_VEL
LIN {X 0,Y 337.19,Z 355.777,A -85,B 0,C 180,E1 13879.577,E2 13879.577} C_VEL
LIN {X 0,Y 333.632,Z 351.136,A -85,B 0,C 180,E1 13877.484,E2 13877.484} C_VEL
LIN {X 0,Y 329.701,Z 346.798,A -85,B 0,C 180,E1 13874.848,E2 13874.848} C_VEL
LIN {X 0,Y 328.566,Z 344.688,A -85,B 0,C 180,E1 13873.91,E2 13873.91} C_VEL
LIN {X 0,Y 325.186,Z 341.777,A -85,B 0,C 180,E1 13870.99,E2 13870.99} C_VEL
LIN {X 0,Y 323.468,Z 338.482,A -85,B 0,C 180,E1 13868.891,E2 13868.891} C_VEL
LIN {X 0,Y 319.773,Z 335.698,A -85,B 0,C 180,E1 13860.717,E2 13860.717} C_VEL
LIN {X 0,Y 320.164,Z 336.219,A -85,B 0,C 180,E1 13856.585,E2 13856.585} C_VEL
LIN {X 0,Y 323.69,Z 338.722,A -85,B 0,C 180,E1 13850.398,E2 13850.398} C_VEL
LIN {X 0,Y 325.539,Z 342.23,A -85,B 0,C 180,E1 13848.215,E2 13848.215} C_VEL
LIN {X 0,Y 328.782,Z 345.074,A -85,B 0,C 180,E1 13845.47,E2 13845.47} C_VEL
LIN {X 0,Y 331.603,Z 349.242,A -85,B 0,C 180,E1 13843.355,E2 13843.355} C_VEL
LIN {X 0,Y 334.745,Z 351.74,A -85,B 0,C 180,E1 13841.452,E2 13841.452} C_VEL
LIN {X 0,Y 337.915,Z 355.666,A -85,B 0,C 180,E1 13839.474,E2 13839.474} C_VEL
LIN {X 0,Y 341.654,Z 358.324,A -85,B 0,C 180,E1 13837.094,E2 13837.094} C_VEL
LIN {X 0,Y 342.971,Z 359.314,A -85,B 0,C 180,E1 13836.186,E2 13836.186} C_VEL
LIN {X 0,Y 345.59,Z 362.607,A -85,B 0,C 180,E1 13834.096,E2 13834.096} C_VEL
LIN {X 0,Y 348.515,Z 364.966,A -85,B 0,C 180,E1 13831.56,E2 13831.56} C_VEL
LIN {X 0,Y 350.921,Z 366.382,A -85,B 0,C 180,E1 13829.24,E2 13829.24} C_VEL
LIN {X 0,Y 353.047,Z 369.757,A -85,B 0,C 180,E1 13826.867,E2 13826.867} C_VEL
LIN {X 0,Y 356.276,Z 372.381,A -85,B 0,C 180,E1 13823.49,E2 13823.49} C_VEL
LIN {X 0,Y 358.05,Z 373.513,A -85,B 0,C 180,E1 13821.587,E2 13821.587} C_VEL
LIN {X 0,Y 360.463,Z 377.108,A -85,B 0,C 180,E1 13818.736,E2 13818.736} C_VEL
LIN {X 0,Y 363.34,Z 379.361,A -85,B 0,C 180,E1 13815.435,E2 13815.435} C_VEL
LIN {X 0,Y 365.276,Z 380.426,A -85,B 0,C 180,E1 13813.18,E2 13813.18} C_VEL
LIN {X 0,Y 367.181,Z 383.578,A -85,B 0,C 180,E1 13810.559,E2 13810.559} C_VEL
LIN {X 0,Y 369.458,Z 385.736,A -85,B 0,C 180,E1 13807.51,E2 13807.51} C_VEL
LIN {X 0,Y 371.95,Z 387.066,A -85,B 0,C 180,E1 13804.111,E2 13804.111} C_VEL
LIN {X 0,Y 372.899,Z 388.045,A -85,B 0,C 180,E1 13802.656,E2 13802.656} C_VEL
LIN {X 0,Y 374.811,Z 391.047,A -85,B 0,C 180,E1 13799.395,E2 13799.395} C_VEL
LIN {X 0,Y 376.834,Z 392.87,A -85,B 0,C 180,E1 13795.794,E2 13795.794} C_VEL
LIN {X 0,Y 378.619,Z 393.845,A -85,B 0,C 180,E1 13792.35,E2 13792.35} C_VEL
LIN {X 0,Y 380.249,Z 394.749,A -85,B 0,C 180,E1 13788.807,E2 13788.807} C_VEL
LIN {X 0,Y 381.368,Z 396.835,A -85,B 0,C 180,E1 13785.246,E2 13785.246} C_VEL
LIN {X 0,Y 382.345,Z 398.271,A -85,B 0,C 180,E1 13781.769,E2 13781.769} C_VEL
LIN {X 0,Y 383.038,Z 399.039,A -85,B 0,C 180,E1 13778.254,E2 13778.254} C_VEL
LIN {X 0,Y 383.593,Z 399.488,A -85,B 0,C 180,E1 13774.635,E2 13774.635} C_VEL
LIN {X 0,Y 383.779,Z 399.654,A -85,B 0,C 180,E1 13771.045,E2 13771.045} C_VEL
LIN {X 0,Y 383.755,Z 399.625,A -85,B 0,C 180,E1 13767.461,E2 13767.461} C_VEL
LIN {X 0,Y 383.386,Z 399.354,A -85,B 0,C 180,E1 13763.862,E2 13763.862} C_VEL
LIN {X 0,Y 382.787,Z 398.776,A -85,B 0,C 180,E1 13760.225,E2 13760.225} C_VEL
LIN {X 0,Y 381.963,Z 397.767,A -85,B 0,C 180,E1 13756.836,E2 13756.836} C_VEL
LIN {X 0,Y 380.981,Z 396.042,A -85,B 0,C 180,E1 13753.318,E2 13753.318} C_VEL
LIN {X 0,Y 379.905,Z 394.505,A -85,B 0,C 180,E1 13750.425,E2 13750.425} C_VEL
LIN {X 0,Y 378.203,Z 393.67,A -85,B 0,C 180,E1 13746.803,E2 13746.803} C_VEL
LIN {X 0,Y 376.125,Z 392.367,A -85,B 0,C 180,E1 13742.94,E2 13742.94} C_VEL
LIN {X 0,Y 374.172,Z 390.181,A -85,B 0,C 180,E1 13739.489,E2 13739.489} C_VEL
LIN {X 0,Y 372.326,Z 387.195,A -85,B 0,C 180,E1 13736.355,E2 13736.355} C_VEL
LIN {X 0,Y 369.766,Z 385.952,A -85,B 0,C 180,E1 13732.91,E2 13732.91} C_VEL
LIN {X 0,Y 367.49,Z 383.933,A -85,B 0,C 180,E1 13729.849,E2 13729.849} C_VEL
LIN {X 0,Y 365.487,Z 380.925,A -85,B 0,C 180,E1 13727.152,E2 13727.152} C_VEL
LIN {X 0,Y 364.87,Z 380.087,A -85,B 0,C 180,E1 13726.327,E2 13726.327} C_VEL
LIN {X 0,Y 361.896,Z 378.421,A -85,B 0,C 180,E1 13722.935,E2 13722.935} C_VEL
LIN {X 0,Y 359.443,Z 375.871,A -85,B 0,C 180,E1 13720.098,E2 13720.098} C_VEL
LIN {X 0,Y 357.621,Z 373.055,A -85,B 0,C 180,E1 13717.958,E2 13717.958} C_VEL
LIN {X 0,Y 354.545,Z 371.198,A -85,B 0,C 180,E1 13714.727,E2 13714.727} C_VEL
LIN {X 0,Y 351.98,Z 368.355,A -85,B 0,C 180,E1 13711.991,E2 13711.991} C_VEL
LIN {X 0,Y 350.676,Z 366.09,A -85,B 0,C 180,E1 13710.499,E2 13710.499} C_VEL
LIN {X 0,Y 347.389,Z 364.223,A -85,B 0,C 180,E1 13707.42,E2 13707.42} C_VEL
LIN {X 0,Y 344.22,Z 361.115,A -85,B 0,C 180,E1 13704.817,E2 13704.817} C_VEL
LIN {X 0,Y 342.399,Z 358.684,A -85,B 0,C 180,E1 13703.399,E2 13703.399} C_VEL
LIN {X 0,Y 338.574,Z 356.25,A -85,B 0,C 180,E1 13700.936,E2 13700.936} C_VEL
LIN {X 0,Y 335.529,Z 352.887,A -85,B 0,C 180,E1 13699.045,E2 13699.045} C_VEL
LIN {X 0,Y 334.043,Z 351.087,A -85,B 0,C 180,E1 13698.137,E2 13698.137} C_VEL
LIN {X 0,Y 330.627,Z 348.117,A -85,B 0,C 180,E1 13695.974,E2 13695.974} C_VEL
LIN {X 0,Y 328.467,Z 344.639,A -85,B 0,C 180,E1 13694.274,E2 13694.274} C_VEL
LIN {X 0,Y 325.032,Z 341.559,A -85,B 0,C 180,E1 13691.264,E2 13691.264} C_VEL
LIN {X 0,Y 323.556,Z 338.496,A -85,B 0,C 180,E1 13689.426,E2 13689.426} C_VEL
LIN {X 0,Y 321.736,Z 337.606,A -85,B 0,C 180,E1 13686.983,E2 13686.983} C_VEL
LIN {X 0,Y 320.798,Z 338.141,A -85,B 0,C 180,E1 13685.512,E2 13685.512} C_VEL
LIN {X 0,Y 318.896,Z 343.265,A -85,B 0,C 180,E1 13681.62,E2 13681.62} C_VEL
LIN {X 0,Y 318.767,Z 343.643,A -85,B 0,C 180,E1 13680.719,E2 13680.719} C_VEL
LIN {X 0,Y 319.31,Z 344.338,A -85,B 0,C 180,E1 13676.589,E2 13676.589} C_VEL
LIN {X 0,Y 322.48,Z 346.627,A -85,B 0,C 180,E1 13671.082,E2 13671.082} C_VEL
LIN {X 0,Y 324.464,Z 350.222,A -85,B 0,C 180,E1 13668.716,E2 13668.716} C_VEL
LIN {X 0,Y 327.4,Z 352.932,A -85,B 0,C 180,E1 13666.174,E2 13666.174} C_VEL
LIN {X 0,Y 330.239,Z 357.053,A -85,B 0,C 180,E1 13664.007,E2 13664.007} C_VEL
LIN {X 0,Y 332.114,Z 358.944,A -85,B 0,C 180,E1 13662.795,E2 13662.795} C_VEL
LIN {X 0,Y 335.778,Z 363.609,A -85,B 0,C 180,E1 13660.609,E2 13660.609} C_VEL
LIN {X 0,Y 341.03,Z 370.717,A -85,B 0,C 180,E1 13657.877,E2 13657.877} C_VEL
LIN {X 0,Y 345.162,Z 376.315,A -85,B 0,C 180,E1 13655.984,E2 13655.984} C_VEL
LIN {X 0,Y 347.777,Z 380.117,A -85,B 0,C 180,E1 13654.863,E2 13654.863} C_VEL
LIN {X 0,Y 354.196,Z 391.08,A -85,B 0,C 180,E1 13652.285,E2 13652.285} C_VEL
LIN {X 0,Y 360.866,Z 403.205,A -85,B 0,C 180,E1 13649.878,E2 13649.878} C_VEL
LIN {X 0,Y 365.938,Z 413.59,A -85,B 0,C 180,E1 13648.169,E2 13648.169} C_VEL
LIN {X 0,Y 354.035,Z 599.94,A -85,B 0,C 180,E1 13644.385,E2 13644.385} C_VEL
LIN {X 0,Y 351.21,Z 623.351,A -85,B 0,C 180,E1 13643.724,E2 13643.724} C_VEL
LIN {X 0,Y 347.856,Z 642.596,A -85,B 0,C 180,E1 13642.972,E2 13642.972} C_VEL
LIN {X 0,Y 343.966,Z 661.026,A -85,B 0,C 180,E1 13642.042,E2 13642.042} C_VEL
LIN {X 0,Y 338.358,Z 683.211,A -85,B 0,C 180,E1 13640.599,E2 13640.599} C_VEL
LIN {X 0,Y 333.364,Z 700.109,A -85,B 0,C 180,E1 13639.227,E2 13639.227} C_VEL
LIN {X 0,Y 328.167,Z 716.09,A -85,B 0,C 180,E1 13637.675,E2 13637.675} C_VEL
LIN {X 0,Y 321.353,Z 735.15,A -85,B 0,C 180,E1 13635.438,E2 13635.438} C_VEL
LIN {X 0,Y 315.335,Z 750.59,A -85,B 0,C 180,E1 13633.225,E2 13633.225} C_VEL
LIN {X 0,Y 309.583,Z 764.684,A -85,B 0,C 180,E1 13630.843,E2 13630.843} C_VEL
LIN {X 0,Y 302.858,Z 780.648,A -85,B 0,C 180,E1 13627.596,E2 13627.596} C_VEL
LIN {X 0,Y 297.601,Z 792.833,A -85,B 0,C 180,E1 13624.595,E2 13624.595} C_VEL
LIN {X 0,Y 293.043,Z 803.634,A -85,B 0,C 180,E1 13621.461,E2 13621.461} C_VEL
LIN {X 0,Y 288.213,Z 815.605,A -85,B 0,C 180,E1 13617.253,E2 13617.253} C_VEL
LIN {X 0,Y 285.069,Z 824.115,A -85,B 0,C 180,E1 13613.568,E2 13613.568} C_VEL
LIN {X 0,Y 282.783,Z 831.243,A -85,B 0,C 180,E1 13609.842,E2 13609.842} C_VEL
LIN {X 0,Y 280.971,Z 838.375,A -85,B 0,C 180,E1 13605.056,E2 13605.056} C_VEL
LIN {X 0,Y 280.266,Z 842.517,A -85,B 0,C 180,E1 13601.315,E2 13601.315} C_VEL
LIN {X 0,Y 280.005,Z 845.347,A -85,B 0,C 180,E1 13597.798,E2 13597.798} C_VEL
LIN {X 0,Y 279.959,Z 847.14,A -85,B 0,C 180,E1 13594.301,E2 13594.301} C_VEL
LIN {X 0,Y 279.971,Z 847.963,A -85,B 0,C 180,E1 13590.409,E2 13590.409} C_VEL
LIN {X 0,Y 279.956,Z 847.388,A -85,B 0,C 180,E1 13586.314,E2 13586.314} C_VEL
LIN {X 0,Y 280,Z 845.486,A -85,B 0,C 180,E1 13582.408,E2 13582.408} C_VEL
LIN {X 0,Y 280.247,Z 842.676,A -85,B 0,C 180,E1 13578.853,E2 13578.853} C_VEL
LIN {X 0,Y 280.916,Z 838.628,A -85,B 0,C 180,E1 13575.152,E2 13575.152} C_VEL
LIN {X 0,Y 282.484,Z 832.356,A -85,B 0,C 180,E1 13570.782,E2 13570.782} C_VEL
LIN {X 0,Y 284.922,Z 824.549,A -85,B 0,C 180,E1 13566.638,E2 13566.638} C_VEL
LIN {X 0,Y 287.817,Z 816.604,A -85,B 0,C 180,E1 13563.154,E2 13563.154} C_VEL
LIN {X 0,Y 292.289,Z 805.54,A -85,B 0,C 180,E1 13559.129,E2 13559.129} C_VEL
LIN {X 0,Y 297.294,Z 793.552,A -85,B 0,C 180,E1 13555.598,E2 13555.598} C_VEL
LIN {X 0,Y 302.215,Z 782.094,A -85,B 0,C 180,E1 13552.74,E2 13552.74} C_VEL
LIN {X 0,Y 308.671,Z 766.968,A -85,B 0,C 180,E1 13549.572,E2 13549.572} C_VEL
LIN {X 0,Y 314.889,Z 751.697,A -85,B 0,C 180,E1 13546.948,E2 13546.948} C_VEL
LIN {X 0,Y 320.64,Z 736.971,A -85,B 0,C 180,E1 13544.808,E2 13544.808} C_VEL
LIN {X 0,Y 327.573,Z 717.888,A -85,B 0,C 180,E1 13542.514,E2 13542.514} C_VEL
LIN {X 0,Y 333.093,Z 700.978,A -85,B 0,C 180,E1 13540.851,E2 13540.851} C_VEL
LIN {X 0,Y 338.074,Z 684.198,A -85,B 0,C 180,E1 13539.476,E2 13539.476} C_VEL
LIN {X 0,Y 343.506,Z 663.141,A -85,B 0,C 180,E1 13538.077,E2 13538.077} C_VEL
LIN {X 0,Y 347.559,Z 644.158,A -85,B 0,C 180,E1 13537.099,E2 13537.099} C_VEL
LIN {X 0,Y 350.731,Z 626.303,A -85,B 0,C 180,E1 13536.382,E2 13536.382} C_VEL
LIN {X 0,Y 353.691,Z 604.067,A -85,B 0,C 180,E1 13535.711,E2 13535.711} C_VEL
LIN {X 0,Y 356.538,Z 562.307,A -85,B 0,C 180,E1 13534.824,E2 13534.824} C_VEL
LIN {X 0,Y 365.904,Z 413.137,A -85,B 0,C 180,E1 13531.806,E2 13531.806} C_VEL
LIN {X 0,Y 357.911,Z 397.697,A -85,B 0,C 180,E1 13529.083,E2 13529.083} C_VEL
LIN {X 0,Y 351.583,Z 386.539,A -85,B 0,C 180,E1 13526.701,E2 13526.701} C_VEL
LIN {X 0,Y 346.334,Z 377.876,A -85,B 0,C 180,E1 13524.519,E2 13524.519} C_VEL
LIN {X 0,Y 342.127,Z 372.223,A -85,B 0,C 180,E1 13522.646,E2 13522.646} C_VEL
LIN {X 0,Y 339.106,Z 368.161,A -85,B 0,C 180,E1 13521.173,E2 13521.173} C_VEL
LIN {X 0,Y 335.327,Z 363.179,A -85,B 0,C 180,E1 13519.147,E2 13519.147} C_VEL
LIN {X 0,Y 331.405,Z 358.06,A -85,B 0,C 180,E1 13516.746,E2 13516.746} C_VEL
LIN {X 0,Y 328.269,Z 354.518,A -85,B 0,C 180,E1 13514.553,E2 13514.553} C_VEL
LIN {X 0,Y 326.934,Z 352.328,A -85,B 0,C 180,E1 13513.44,E2 13513.44} C_VEL
LIN {X 0,Y 323.56,Z 348.992,A -85,B 0,C 180,E1 13510.325,E2 13510.325} C_VEL
LIN {X 0,Y 322.208,Z 346.301,A -85,B 0,C 180,E1 13508.566,E2 13508.566} C_VEL
LIN {X 0,Y 318.797,Z 343.642,A -85,B 0,C 180,E1 13500.719,E2 13500.719} C_VEL
LIN {X 0,Y 319.188,Z 344.176,A -85,B 0,C 180,E1 13496.576,E2 13496.576} C_VEL
LIN {X 0,Y 322.492,Z 346.623,A -85,B 0,C 180,E1 13490.632,E2 13490.632} C_VEL
LIN {X 0,Y 324.477,Z 350.235,A -85,B 0,C 180,E1 13488.266,E2 13488.266} C_VEL
LIN {X 0,Y 327.369,Z 352.847,A -85,B 0,C 180,E1 13485.767,E2 13485.767} C_VEL
LIN {X 0,Y 330.387,Z 357.18,A -85,B 0,C 180,E1 13483.473,E2 13483.473} C_VEL
LIN {X 0,Y 333.217,Z 359.496,A -85,B 0,C 180,E1 13481.726,E2 13481.726} C_VEL
LIN {X 0,Y 336.571,Z 363.49,A -85,B 0,C 180,E1 13479.661,E2 13479.661} C_VEL
LIN {X 0,Y 340.292,Z 366.124,A -85,B 0,C 180,E1 13477.306,E2 13477.306} C_VEL
LIN {X 0,Y 341.568,Z 367.06,A -85,B 0,C 180,E1 13476.449,E2 13476.449} C_VEL
LIN {X 0,Y 344.449,Z 370.54,A -85,B 0,C 180,E1 13474.188,E2 13474.188} C_VEL
LIN {X 0,Y 347.416,Z 372.872,A -85,B 0,C 180,E1 13471.649,E2 13471.649} C_VEL
LIN {X 0,Y 349.793,Z 374.381,A -85,B 0,C 180,E1 13469.357,E2 13469.357} C_VEL
LIN {X 0,Y 351.983,Z 377.714,A -85,B 0,C 180,E1 13466.926,E2 13466.926} C_VEL
LIN {X 0,Y 355.208,Z 380.296,A -85,B 0,C 180,E1 13463.564,E2 13463.564} C_VEL
LIN {X 0,Y 356.892,Z 381.403,A -85,B 0,C 180,E1 13461.746,E2 13461.746} C_VEL
LIN {X 0,Y 359.29,Z 384.918,A -85,B 0,C 180,E1 13458.947,E2 13458.947} C_VEL
LIN {X 0,Y 362.305,Z 387.285,A -85,B 0,C 180,E1 13455.496,E2 13455.496} C_VEL
LIN {X 0,Y 364.186,Z 388.35,A -85,B 0,C 180,E1 13453.319,E2 13453.319} C_VEL
LIN {X 0,Y 366.218,Z 391.608,A -85,B 0,C 180,E1 13450.525,E2 13450.525} C_VEL
LIN {X 0,Y 368.578,Z 393.769,A -85,B 0,C 180,E1 13447.361,E2 13447.361} C_VEL
LIN {X 0,Y 371.142,Z 395.065,A -85,B 0,C 180,E1 13443.893,E2 13443.893} C_VEL
LIN {X 0,Y 371.975,Z 396.263,A -85,B 0,C 180,E1 13442.519,E2 13442.519} C_VEL
LIN {X 0,Y 373.886,Z 399.078,A -85,B 0,C 180,E1 13439.299,E2 13439.299} C_VEL
LIN {X 0,Y 375.932,Z 400.885,A -85,B 0,C 180,E1 13435.627,E2 13435.627} C_VEL
LIN {X 0,Y 377.695,Z 401.808,A -85,B 0,C 180,E1 13432.244,E2 13432.244} C_VEL
LIN {X 0,Y 379.283,Z 402.721,A -85,B 0,C 180,E1 13428.76,E2 13428.76} C_VEL
LIN {X 0,Y 380.378,Z 404.778,A -85,B 0,C 180,E1 13425.271,E2 13425.271} C_VEL
LIN {X 0,Y 381.362,Z 406.208,A -85,B 0,C 180,E1 13421.8,E2 13421.8} C_VEL
LIN {X 0,Y 382.057,Z 406.978,A -85,B 0,C 180,E1 13418.276,E2 13418.276} C_VEL
LIN {X 0,Y 382.619,Z 407.428,A -85,B 0,C 180,E1 13414.646,E2 13414.646} C_VEL
LIN {X 0,Y 382.802,Z 407.594,A -85,B 0,C 180,E1 13411.048,E2 13411.048} C_VEL
LIN {X 0,Y 382.782,Z 407.566,A -85,B 0,C 180,E1 13407.455,E2 13407.455} C_VEL
LIN {X 0,Y 382.422,Z 407.32,A -85,B 0,C 180,E1 13403.997,E2 13403.997} C_VEL
LIN {X 0,Y 381.847,Z 406.748,A -85,B 0,C 180,E1 13400.353,E2 13400.353} C_VEL
LIN {X 0,Y 380.979,Z 405.709,A -85,B 0,C 180,E1 13396.822,E2 13396.822} C_VEL
LIN {X 0,Y 379.991,Z 404.005,A -85,B 0,C 180,E1 13393.291,E2 13393.291} C_VEL
LIN {X 0,Y 378.916,Z 402.444,A -85,B 0,C 180,E1 13390.394,E2 13390.394} C_VEL
LIN {X 0,Y 377.192,Z 401.596,A -85,B 0,C 180,E1 13386.737,E2 13386.737} C_VEL
LIN {X 0,Y 375.109,Z 400.294,A -85,B 0,C 180,E1 13382.884,E2 13382.884} C_VEL
LIN {X 0,Y 373.13,Z 398.095,A -85,B 0,C 180,E1 13379.395,E2 13379.395} C_VEL
LIN {X 0,Y 371.309,Z 395.126,A -85,B 0,C 180,E1 13376.31,E2 13376.31} C_VEL
LIN {X 0,Y 368.688,Z 393.846,A -85,B 0,C 180,E1 13372.789,E2 13372.789} C_VEL
LIN {X 0,Y 366.311,Z 391.714,A -85,B 0,C 180,E1 13369.6,E2 13369.6} C_VEL
LIN {X 0,Y 364.313,Z 388.659,A -85,B 0,C 180,E1 13366.889,E2 13366.889} C_VEL
LIN {X 0,Y 363.656,Z 387.948,A -85,B 0,C 180,E1 13366.084,E2 13366.084} C_VEL
LIN {X 0,Y 360.727,Z 386.251,A -85,B 0,C 180,E1 13362.735,E2 13362.735} C_VEL
LIN {X 0,Y 358.25,Z 383.653,A -85,B 0,C 180,E1 13359.871,E2 13359.871} C_VEL
LIN {X 0,Y 356.386,Z 380.893,A -85,B 0,C 180,E1 13357.706,E2 13357.706} C_VEL
LIN {X 0,Y 353.322,Z 378.975,A -85,B 0,C 180,E1 13354.47,E2 13354.47} C_VEL
LIN {X 0,Y 350.657,Z 375.97,A -85,B 0,C 180,E1 13351.645,E2 13351.645} C_VEL
LIN {X 0,Y 349.366,Z 373.912,A -85,B 0,C 180,E1 13350.2,E2 13350.2} C_VEL
LIN {X 0,Y 346.036,Z 371.962,A -85,B 0,C 180,E1 13347.136,E2 13347.136} C_VEL
LIN {X 0,Y 342.83,Z 368.839,A -85,B 0,C 180,E1 13344.557,E2 13344.557} C_VEL
LIN {X 0,Y 340.976,Z 366.46,A -85,B 0,C 180,E1 13343.137,E2 13343.137} C_VEL
LIN {X 0,Y 337.098,Z 363.955,A -85,B 0,C 180,E1 13340.669,E2 13340.669} C_VEL
LIN {X 0,Y 333.754,Z 360.257,A -85,B 0,C 180,E1 13338.606,E2 13338.606} C_VEL
LIN {X 0,Y 332.532,Z 358.805,A -85,B 0,C 180,E1 13337.86,E2 13337.86} C_VEL
LIN {X 0,Y 329.051,Z 355.644,A -85,B 0,C 180,E1 13335.589,E2 13335.589} C_VEL
LIN {X 0,Y 327.062,Z 352.398,A -85,B 0,C 180,E1 13333.976,E2 13333.976} C_VEL
LIN {X 0,Y 323.649,Z 349.128,A -85,B 0,C 180,E1 13330.862,E2 13330.862} C_VEL
LIN {X 0,Y 322.294,Z 346.313,A -85,B 0,C 180,E1 13329.103,E2 13329.103} C_VEL
LIN {X 0,Y 318.791,Z 343.641,A -85,B 0,C 180,E1 13321.078,E2 13321.078} C_VEL
LIN {X 0,Y 318.767,Z 343.643,A -85,B 0,C 180,E1 13320.719,E2 13320.719} C_VEL
LIN {X 0,Y 318.657,Z 344.746,A -85,B 0,C 180,E1 13319.338,E2 13319.338} C_VEL
LIN {X 0,Y 318.768,Z 352.213,A -85,B 0,C 180,E1 13315.532,E2 13315.532} C_VEL
LIN {X 0,Y 319.156,Z 353.116,A -85,B 0,C 180,E1 13314.544,E2 13314.544} C_VEL
LIN {X 0,Y 321.288,Z 354.51,A -85,B 0,C 180,E1 13311.319,E2 13311.319} C_VEL
LIN {X 0,Y 323.401,Z 358.222,A -85,B 0,C 180,E1 13308.768,E2 13308.768} C_VEL
LIN {X 0,Y 325.947,Z 360.588,A -85,B 0,C 180,E1 13306.518,E2 13306.518} C_VEL
LIN {X 0,Y 328.9,Z 364.862,A -85,B 0,C 180,E1 13304.212,E2 13304.212} C_VEL
LIN {X 0,Y 330.545,Z 366.625,A -85,B 0,C 180,E1 13303.119,E2 13303.119} C_VEL
LIN {X 0,Y 334.844,Z 372.401,A -85,B 0,C 180,E1 13300.507,E2 13300.507} C_VEL
LIN {X 0,Y 339.075,Z 378.117,A -85,B 0,C 180,E1 13298.28,E2 13298.28} C_VEL
LIN {X 0,Y 343.46,Z 384.193,A -85,B 0,C 180,E1 13296.222,E2 13296.222} C_VEL
LIN {X 0,Y 345.665,Z 387.634,A -85,B 0,C 180,E1 13295.248,E2 13295.248} C_VEL
LIN {X 0,Y 351.488,Z 397.83,A -85,B 0,C 180,E1 13292.834,E2 13292.834} C_VEL
LIN {X 0,Y 357.754,Z 409.515,A -85,B 0,C 180,E1 13290.489,E2 13290.489} C_VEL
LIN {X 0,Y 361.492,Z 417.336,A -85,B 0,C 180,E1 13289.171,E2 13289.171} C_VEL
LIN {X 0,Y 349.409,Z 599.804,A -85,B 0,C 180,E1 13285.453,E2 13285.453} C_VEL
LIN {X 0,Y 346.444,Z 623.507,A -85,B 0,C 180,E1 13284.782,E2 13284.782} C_VEL
LIN {X 0,Y 343.007,Z 642.619,A -85,B 0,C 180,E1 13284.035,E2 13284.035} C_VEL
LIN {X 0,Y 338.903,Z 661.439,A -85,B 0,C 180,E1 13283.083,E2 13283.083} C_VEL
LIN {X 0,Y 333.265,Z 682.959,A -85,B 0,C 180,E1 13281.677,E2 13281.677} C_VEL
LIN {X 0,Y 328.199,Z 699.557,A -85,B 0,C 180,E1 13280.331,E2 13280.331} C_VEL
LIN {X 0,Y 322.897,Z 715.321,A -85,B 0,C 180,E1 13278.802,E2 13278.802} C_VEL
LIN {X 0,Y 316.152,Z 733.677,A -85,B 0,C 180,E1 13276.664,E2 13276.664} C_VEL
LIN {X 0,Y 309.393,Z 750.335,A -85,B 0,C 180,E1 13274.269,E2 13274.269} C_VEL
LIN {X 0,Y 303.602,Z 763.93,A -85,B 0,C 180,E1 13271.953,E2 13271.953} C_VEL
LIN {X 0,Y 296.789,Z 779.428,A -85,B 0,C 180,E1 13268.8,E2 13268.8} C_VEL
LIN {X 0,Y 291.145,Z 791.857,A -85,B 0,C 180,E1 13265.718,E2 13265.718} C_VEL
LIN {X 0,Y 286.281,Z 802.718,A -85,B 0,C 180,E1 13262.537,E2 13262.537} C_VEL
LIN {X 0,Y 281.53,Z 813.848,A -85,B 0,C 180,E1 13258.649,E2 13258.649} C_VEL
LIN {X 0,Y 277.668,Z 823.424,A -85,B 0,C 180,E1 13254.462,E2 13254.462} C_VEL
LIN {X 0,Y 275.281,Z 830.244,A -85,B 0,C 180,E1 13250.851,E2 13250.851} C_VEL
LIN {X 0,Y 273.34,Z 837.106,A -85,B 0,C 180,E1 13246.359,E2 13246.359} C_VEL
LIN {X 0,Y 272.332,Z 842.069,A -85,B 0,C 180,E1 13241.864,E2 13241.864} C_VEL
LIN {X 0,Y 272.028,Z 844.957,A -85,B 0,C 180,E1 13238.241,E2 13238.241} C_VEL
LIN {X 0,Y 271.962,Z 846.808,A -85,B 0,C 180,E1 13234.639,E2 13234.639} C_VEL
LIN {X 0,Y 271.975,Z 847.633,A -85,B 0,C 180,E1 13231.053,E2 13231.053} C_VEL
LIN {X 0,Y 271.964,Z 847.382,A -85,B 0,C 180,E1 13227.05,E2 13227.05} C_VEL
LIN {X 0,Y 271.997,Z 845.513,A -85,B 0,C 180,E1 13222.608,E2 13222.608} C_VEL
LIN {X 0,Y 272.267,Z 842.559,A -85,B 0,C 180,E1 13218.671,E2 13218.671} C_VEL
LIN {X 0,Y 272.966,Z 838.627,A -85,B 0,C 180,E1 13214.926,E2 13214.926} C_VEL
LIN {X 0,Y 274.621,Z 832.454,A -85,B 0,C 180,E1 13210.431,E2 13210.431} C_VEL
LIN {X 0,Y 277.194,Z 824.726,A -85,B 0,C 180,E1 13206.173,E2 13206.173} C_VEL
LIN {X 0,Y 280.242,Z 816.846,A -85,B 0,C 180,E1 13202.597,E2 13202.597} C_VEL
LIN {X 0,Y 284.671,Z 806.489,A -85,B 0,C 180,E1 13198.681,E2 13198.681} C_VEL
LIN {X 0,Y 290.17,Z 794.013,A -85,B 0,C 180,E1 13194.87,E2 13194.87} C_VEL
LIN {X 0,Y 295.302,Z 782.64,A -85,B 0,C 180,E1 13191.96,E2 13191.96} C_VEL
LIN {X 0,Y 301.934,Z 767.9,A -85,B 0,C 180,E1 13188.778,E2 13188.778} C_VEL
LIN {X 0,Y 308.468,Z 752.549,A -85,B 0,C 180,E1 13186.082,E2 13186.082} C_VEL
LIN {X 0,Y 314.429,Z 737.915,A -85,B 0,C 180,E1 13183.913,E2 13183.913} C_VEL
LIN {X 0,Y 321.32,Z 719.945,A -85,B 0,C 180,E1 13181.687,E2 13181.687} C_VEL
LIN {X 0,Y 327.547,Z 701.595,A -85,B 0,C 180,E1 13179.852,E2 13179.852} C_VEL
LIN {X 0,Y 332.39,Z 685.92,A -85,B 0,C 180,E1 13178.549,E2 13178.549} C_VEL
LIN {X 0,Y 337.41,Z 667.619,A -85,B 0,C 180,E1 13177.285,E2 13177.285} C_VEL
LIN {X 0,Y 342.292,Z 646.283,A -85,B 0,C 180,E1 13176.133,E2 13176.133} C_VEL
LIN {X 0,Y 345.717,Z 627.875,A -85,B 0,C 180,E1 13175.375,E2 13175.375} C_VEL
LIN {X 0,Y 348.491,Z 608.621,A -85,B 0,C 180,E1 13174.771,E2 13174.771} C_VEL
LIN {X 0,Y 350.899,Z 579.525,A -85,B 0,C 180,E1 13174.106,E2 13174.106} C_VEL
LIN {X 0,Y 361.454,Z 417.008,A -85,B 0,C 180,E1 13170.806,E2 13170.806} C_VEL
LIN {X 0,Y 354.52,Z 403.363,A -85,B 0,C 180,E1 13168.328,E2 13168.328} C_VEL
LIN {X 0,Y 348.659,Z 392.783,A -85,B 0,C 180,E1 13166.025,E2 13166.025} C_VEL
LIN {X 0,Y 343.904,Z 384.785,A -85,B 0,C 180,E1 13163.973,E2 13163.973} C_VEL
LIN {X 0,Y 339.56,Z 378.809,A -85,B 0,C 180,E1 13161.96,E2 13161.96} C_VEL
LIN {X 0,Y 336.863,Z 375.162,A -85,B 0,C 180,E1 13160.593,E2 13160.593} C_VEL
LIN {X 0,Y 333.34,Z 370.425,A -85,B 0,C 180,E1 13158.63,E2 13158.63} C_VEL
LIN {X 0,Y 329.789,Z 365.653,A -85,B 0,C 180,E1 13156.377,E2 13156.377} C_VEL
LIN {X 0,Y 326.639,Z 361.886,A -85,B 0,C 180,E1 13154.084,E2 13154.084} C_VEL
LIN {X 0,Y 325.541,Z 360.075,A -85,B 0,C 180,E1 13153.137,E2 13153.137} C_VEL
LIN {X 0,Y 322.198,Z 356.553,A -85,B 0,C 180,E1 13149.917,E2 13149.917} C_VEL
LIN {X 0,Y 321.098,Z 354.193,A -85,B 0,C 180,E1 13148.416,E2 13148.416} C_VEL
LIN {X 0,Y 317.822,Z 351.587,A -85,B 0,C 180,E1 13140.721,E2 13140.721} C_VEL
LIN {X 0,Y 318.212,Z 352.134,A -85,B 0,C 180,E1 13136.568,E2 13136.568} C_VEL
LIN {X 0,Y 321.3,Z 354.509,A -85,B 0,C 180,E1 13130.868,E2 13130.868} C_VEL
LIN {X 0,Y 323.329,Z 358.134,A -85,B 0,C 180,E1 13128.404,E2 13128.404} C_VEL
LIN {X 0,Y 325.966,Z 360.601,A -85,B 0,C 180,E1 13126.067,E2 13126.067} C_VEL
LIN {X 0,Y 329.048,Z 364.991,A -85,B 0,C 180,E1 13123.676,E2 13123.676} C_VEL
LIN {X 0,Y 331.698,Z 367.244,A -85,B 0,C 180,E1 13122.003,E2 13122.003} C_VEL
LIN {X 0,Y 335.36,Z 371.429,A -85,B 0,C 180,E1 13119.766,E2 13119.766} C_VEL
LIN {X 0,Y 339.283,Z 374.105,A -85,B 0,C 180,E1 13117.291,E2 13117.291} C_VEL
LIN {X 0,Y 340.489,Z 375.272,A -85,B 0,C 180,E1 13116.461,E2 13116.461} C_VEL
LIN {X 0,Y 343.596,Z 378.746,A -85,B 0,C 180,E1 13114.048,E2 13114.048} C_VEL
LIN {X 0,Y 346.699,Z 380.995,A -85,B 0,C 180,E1 13111.397,E2 13111.397} C_VEL
LIN {X 0,Y 348.574,Z 382.188,A -85,B 0,C 180,E1 13109.584,E2 13109.584} C_VEL
LIN {X 0,Y 350.709,Z 385.451,A -85,B 0,C 180,E1 13107.202,E2 13107.202} C_VEL
LIN {X 0,Y 353.777,Z 388.024,A -85,B 0,C 180,E1 13103.995,E2 13103.995} C_VEL
LIN {X 0,Y 355.743,Z 389.3,A -85,B 0,C 180,E1 13101.901,E2 13101.901} C_VEL
LIN {X 0,Y 358.076,Z 392.708,A -85,B 0,C 180,E1 13099.174,E2 13099.174} C_VEL
LIN {X 0,Y 361.093,Z 395.117,A -85,B 0,C 180,E1 13095.751,E2 13095.751} C_VEL
LIN {X 0,Y 363.061,Z 396.242,A -85,B 0,C 180,E1 13093.475,E2 13093.475} C_VEL
LIN {X 0,Y 365.127,Z 399.482,A -85,B 0,C 180,E1 13090.665,E2 13090.665} C_VEL
LIN {X 0,Y 367.452,Z 401.626,A -85,B 0,C 180,E1 13087.553,E2 13087.553} C_VEL
LIN {X 0,Y 369.914,Z 402.926,A -85,B 0,C 180,E1 13084.198,E2 13084.198} C_VEL
LIN {X 0,Y 370.721,Z 403.761,A -85,B 0,C 180,E1 13082.988,E2 13082.988} C_VEL
LIN {X 0,Y 372.604,Z 406.738,A -85,B 0,C 180,E1 13079.764,E2 13079.764} C_VEL
LIN {X 0,Y 374.648,Z 408.579,A -85,B 0,C 180,E1 13076.271,E2 13076.271} C_VEL
LIN {X 0,Y 376.501,Z 409.673,A -85,B 0,C 180,E1 13072.647,E2 13072.647} C_VEL
LIN {X 0,Y 378.143,Z 410.539,A -85,B 0,C 180,E1 13069.139,E2 13069.139} C_VEL
LIN {X 0,Y 379.295,Z 412.59,A -85,B 0,C 180,E1 13065.597,E2 13065.597} C_VEL
LIN {X 0,Y 380.3,Z 414.042,A -85,B 0,C 180,E1 13062.141,E2 13062.141} C_VEL
LIN {X 0,Y 381.029,Z 414.847,A -85,B 0,C 180,E1 13058.602,E2 13058.602} C_VEL
LIN {X 0,Y 381.568,Z 415.317,A -85,B 0,C 180,E1 13055.262,E2 13055.262} C_VEL
LIN {X 0,Y 381.816,Z 415.551,A -85,B 0,C 180,E1 13051.651,E2 13051.651} C_VEL
LIN {X 0,Y 381.816,Z 415.551,A -85,B 0,C 180,E1 13048.349,E2 13048.349} C_VEL
LIN {X 0,Y 381.536,Z 415.312,A -85,B 0,C 180,E1 13044.587,E2 13044.587} C_VEL
LIN {X 0,Y 381.008,Z 414.818,A -85,B 0,C 180,E1 13041.245,E2 13041.245} C_VEL
LIN {X 0,Y 380.212,Z 413.922,A -85,B 0,C 180,E1 13037.547,E2 13037.547} C_VEL
LIN {X 0,Y 379.242,Z 412.509,A -85,B 0,C 180,E1 13034.218,E2 13034.218} C_VEL
LIN {X 0,Y 378.068,Z 410.493,A -85,B 0,C 180,E1 13030.696,E2 13030.696} C_VEL
LIN {X 0,Y 376.501,Z 409.674,A -85,B 0,C 180,E1 13027.353,E2 13027.353} C_VEL
LIN {X 0,Y 374.647,Z 408.579,A -85,B 0,C 180,E1 13023.729,E2 13023.729} C_VEL
LIN {X 0,Y 372.604,Z 406.738,A -85,B 0,C 180,E1 13020.236,E2 13020.236} C_VEL
LIN {X 0,Y 370.721,Z 403.762,A -85,B 0,C 180,E1 13017.012,E2 13017.012} C_VEL
LIN {X 0,Y 369.906,Z 402.923,A -85,B 0,C 180,E1 13015.791,E2 13015.791} C_VEL
LIN {X 0,Y 367.396,Z 401.585,A -85,B 0,C 180,E1 13012.368,E2 13012.368} C_VEL
LIN {X 0,Y 364.96,Z 399.274,A -85,B 0,C 180,E1 13009.099,E2 13009.099} C_VEL
LIN {X 0,Y 362.8,Z 395.94,A -85,B 0,C 180,E1 13006.224,E2 13006.224} C_VEL
LIN {X 0,Y 359.797,Z 394.279,A -85,B 0,C 180,E1 13002.809,E2 13002.809} C_VEL
LIN {X 0,Y 357.162,Z 391.586,A -85,B 0,C 180,E1 12999.767,E2 12999.767} C_VEL
LIN {X 0,Y 355.327,Z 388.81,A -85,B 0,C 180,E1 12997.634,E2 12997.634} C_VEL
LIN {X 0,Y 352.152,Z 386.813,A -85,B 0,C 180,E1 12994.289,E2 12994.289} C_VEL
LIN {X 0,Y 349.422,Z 383.713,A -85,B 0,C 180,E1 12991.385,E2 12991.385} C_VEL
LIN {X 0,Y 348.142,Z 381.764,A -85,B 0,C 180,E1 12989.982,E2 12989.982} C_VEL
LIN {X 0,Y 344.747,Z 379.742,A -85,B 0,C 180,E1 12986.9,E2 12986.9} C_VEL
LIN {X 0,Y 341.45,Z 376.563,A -85,B 0,C 180,E1 12984.294,E2 12984.294} C_VEL
LIN {X 0,Y 339.539,Z 374.229,A -85,B 0,C 180,E1 12982.874,E2 12982.874} C_VEL
LIN {X 0,Y 335.621,Z 371.658,A -85,B 0,C 180,E1 12980.399,E2 12980.399} C_VEL
LIN {X 0,Y 332.093,Z 367.807,A -85,B 0,C 180,E1 12978.247,E2 12978.247} C_VEL
LIN {X 0,Y 330.752,Z 366.342,A -85,B 0,C 180,E1 12977.414,E2 12977.414} C_VEL
LIN {X 0,Y 327.296,Z 362.896,A -85,B 0,C 180,E1 12975.05,E2 12975.05} C_VEL
LIN {X 0,Y 325.668,Z 360.149,A -85,B 0,C 180,E1 12973.674,E2 12973.674} C_VEL
LIN {X 0,Y 322.276,Z 356.682,A -85,B 0,C 180,E1 12970.448,E2 12970.448} C_VEL
LIN {X 0,Y 321.041,Z 354.147,A -85,B 0,C 180,E1 12968.778,E2 12968.778} C_VEL
LIN {X 0,Y 317.816,Z 351.582,A -85,B 0,C 180,E1 12961.082,E2 12961.082} C_VEL
LIN {X 0,Y 318.182,Z 352.1,A -85,B 0,C 180,E1 12957.118,E2 12957.118} C_VEL
LIN {X 0,Y 319.156,Z 353.116,A -85,B 0,C 180,E1 12954.544,E2 12954.544} C_VEL
LIN {X 0,Y 319.698,Z 354.483,A -85,B 0,C 180,E1 12953.379,E2 12953.379} C_VEL
LIN {X 0,Y 320.406,Z 358.692,A -85,B 0,C 180,E1 12951.743,E2 12951.743} C_VEL
LIN {X 0,Y 321.671,Z 364.826,A -85,B 0,C 180,E1 12949.591,E2 12949.591} C_VEL
LIN {X 0,Y 322.518,Z 366.413,A -85,B 0,C 180,E1 12948.643,E2 12948.643} C_VEL
LIN {X 0,Y 324.554,Z 368.334,A -85,B 0,C 180,E1 12946.822,E2 12946.822} C_VEL
LIN {X 0,Y 327.566,Z 372.671,A -85,B 0,C 180,E1 12944.418,E2 12944.418} C_VEL
LIN {X 0,Y 328.987,Z 374.297,A -85,B 0,C 180,E1 12943.446,E2 12943.446} C_VEL
LIN {X 0,Y 333.129,Z 379.991,A -85,B 0,C 180,E1 12940.858,E2 12940.858} C_VEL
LIN {X 0,Y 337.201,Z 385.607,A -85,B 0,C 180,E1 12938.656,E2 12938.656} C_VEL
LIN {X 0,Y 342.294,Z 392.761,A -85,B 0,C 180,E1 12936.228,E2 12936.228} C_VEL
LIN {X 0,Y 348.72,Z 404.398,A -85,B 0,C 180,E1 12933.43,E2 12933.43} C_VEL
LIN {X 0,Y 354.684,Z 415.826,A -85,B 0,C 180,E1 12931.111,E2 12931.111} C_VEL
LIN {X 0,Y 357.148,Z 421.249,A -85,B 0,C 180,E1 12930.195,E2 12930.195} C_VEL
LIN {X 0,Y 344.916,Z 599.567,A -85,B 0,C 180,E1 12926.553,E2 12926.553} C_VEL
LIN {X 0,Y 341.839,Z 623.434,A -85,B 0,C 180,E1 12925.877,E2 12925.877} C_VEL
LIN {X 0,Y 338.386,Z 642.115,A -85,B 0,C 180,E1 12925.152,E2 12925.152} C_VEL
LIN {X 0,Y 334.265,Z 660.529,A -85,B 0,C 180,E1 12924.227,E2 12924.227} C_VEL
LIN {X 0,Y 328.302,Z 682.683,A -85,B 0,C 180,E1 12922.79,E2 12922.79} C_VEL
LIN {X 0,Y 322.963,Z 699.603,A -85,B 0,C 180,E1 12921.415,E2 12921.415} C_VEL
LIN {X 0,Y 317.302,Z 715.838,A -85,B 0,C 180,E1 12919.829,E2 12919.829} C_VEL
LIN {X 0,Y 309.805,Z 735.257,A -85,B 0,C 180,E1 12917.513,E2 12917.513} C_VEL
LIN {X 0,Y 303.427,Z 750.38,A -85,B 0,C 180,E1 12915.304,E2 12915.304} C_VEL
LIN {X 0,Y 297.298,Z 764.171,A -85,B 0,C 180,E1 12912.923,E2 12912.923} C_VEL
LIN {X 0,Y 289.988,Z 779.974,A -85,B 0,C 180,E1 12909.632,E2 12909.632} C_VEL
LIN {X 0,Y 284.112,Z 792.318,A -85,B 0,C 180,E1 12906.494,E2 12906.494} C_VEL
LIN {X 0,Y 279.03,Z 803.101,A -85,B 0,C 180,E1 12903.246,E2 12903.246} C_VEL
LIN {X 0,Y 273.579,Z 815.09,A -85,B 0,C 180,E1 12898.843,E2 12898.843} C_VEL
LIN {X 0,Y 269.986,Z 823.601,A -85,B 0,C 180,E1 12894.972,E2 12894.972} C_VEL
LIN {X 0,Y 267.344,Z 830.731,A -85,B 0,C 180,E1 12891.04,E2 12891.04} C_VEL
LIN {X 0,Y 265.207,Z 837.867,A -85,B 0,C 180,E1 12885.975,E2 12885.975} C_VEL
LIN {X 0,Y 264.348,Z 842.012,A -85,B 0,C 180,E1 12882.007,E2 12882.007} C_VEL
LIN {X 0,Y 264.03,Z 844.846,A -85,B 0,C 180,E1 12878.274,E2 12878.274} C_VEL
LIN {X 0,Y 263.963,Z 846.642,A -85,B 0,C 180,E1 12874.562,E2 12874.562} C_VEL
LIN {X 0,Y 263.979,Z 847.466,A -85,B 0,C 180,E1 12870.434,E2 12870.434} C_VEL
LIN {X 0,Y 263.962,Z 846.891,A -85,B 0,C 180,E1 12866.091,E2 12866.091} C_VEL
LIN {X 0,Y 264.019,Z 844.985,A -85,B 0,C 180,E1 12861.945,E2 12861.945} C_VEL
LIN {X 0,Y 264.319,Z 842.208,A -85,B 0,C 180,E1 12858.214,E2 12858.214} C_VEL
LIN {X 0,Y 265.143,Z 838.12,A -85,B 0,C 180,E1 12854.246,E2 12854.246} C_VEL
LIN {X 0,Y 267.107,Z 831.474,A -85,B 0,C 180,E1 12849.399,E2 12849.399} C_VEL
LIN {X 0,Y 269.85,Z 823.945,A -85,B 0,C 180,E1 12845.2,E2 12845.2} C_VEL
LIN {X 0,Y 273.352,Z 815.59,A -85,B 0,C 180,E1 12841.37,E2 12841.37} C_VEL
LIN {X 0,Y 278.74,Z 803.742,A -85,B 0,C 180,E1 12836.96,E2 12836.96} C_VEL
LIN {X 0,Y 283.77,Z 793.037,A -85,B 0,C 180,E1 12833.706,E2 12833.706} C_VEL
LIN {X 0,Y 289.224,Z 781.555,A -85,B 0,C 180,E1 12830.748,E2 12830.748} C_VEL
LIN {X 0,Y 296.359,Z 766.296,A -85,B 0,C 180,E1 12827.47,E2 12827.47} C_VEL
LIN {X 0,Y 303.075,Z 751.186,A -85,B 0,C 180,E1 12824.824,E2 12824.824} C_VEL
LIN {X 0,Y 309.286,Z 736.489,A -85,B 0,C 180,E1 12822.656,E2 12822.656} C_VEL
LIN {X 0,Y 316.832,Z 717.165,A -85,B 0,C 180,E1 12820.311,E2 12820.311} C_VEL
LIN {X 0,Y 322.675,Z 700.472,A -85,B 0,C 180,E1 12818.663,E2 12818.663} C_VEL
LIN {X 0,Y 327.994,Z 683.694,A -85,B 0,C 180,E1 12817.287,E2 12817.287} C_VEL
LIN {X 0,Y 333.803,Z 662.507,A -85,B 0,C 180,E1 12815.883,E2 12815.883} C_VEL
LIN {X 0,Y 338.016,Z 643.952,A -85,B 0,C 180,E1 12814.932,E2 12814.932} C_VEL
LIN {X 0,Y 341.417,Z 625.906,A -85,B 0,C 180,E1 12814.212,E2 12814.212} C_VEL
LIN {X 0,Y 344.549,Z 603.672,A -85,B 0,C 180,E1 12813.544,E2 12813.544} C_VEL
LIN {X 0,Y 347.586,Z 562.19,A -85,B 0,C 180,E1 12812.657,E2 12812.657} C_VEL
LIN {X 0,Y 357.117,Z 420.787,A -85,B 0,C 180,E1 12809.778,E2 12809.778} C_VEL
LIN {X 0,Y 350.62,Z 407.893,A -85,B 0,C 180,E1 12807.33,E2 12807.33} C_VEL
LIN {X 0,Y 344.72,Z 397.061,A -85,B 0,C 180,E1 12804.871,E2 12804.871} C_VEL
LIN {X 0,Y 341.333,Z 391.452,A -85,B 0,C 180,E1 12803.34,E2 12803.34} C_VEL
LIN {X 0,Y 335.735,Z 383.425,A -85,B 0,C 180,E1 12800.574,E2 12800.574} C_VEL
LIN {X 0,Y 331.521,Z 377.815,A -85,B 0,C 180,E1 12798.189,E2 12798.189} C_VEL
LIN {X 0,Y 328.189,Z 373.239,A -85,B 0,C 180,E1 12796.005,E2 12796.005} C_VEL
LIN {X 0,Y 325.032,Z 369.253,A -85,B 0,C 180,E1 12793.611,E2 12793.611} C_VEL
LIN {X 0,Y 324.158,Z 367.816,A -85,B 0,C 180,E1 12792.831,E2 12792.831} C_VEL
LIN {X 0,Y 320.852,Z 364.113,A -85,B 0,C 180,E1 12789.507,E2 12789.507} C_VEL
LIN {X 0,Y 319.852,Z 362.023,A -85,B 0,C 180,E1 12788.087,E2 12788.087} C_VEL
LIN {X 0,Y 316.834,Z 359.509,A -85,B 0,C 180,E1 12780.542,E2 12780.542} C_VEL
LIN {X 0,Y 317.284,Z 360.154,A -85,B 0,C 180,E1 12776.386,E2 12776.386} C_VEL
LIN {X 0,Y 320.117,Z 362.38,A -85,B 0,C 180,E1 12771.106,E2 12771.106} C_VEL
LIN {X 0,Y 322.182,Z 366.032,A -85,B 0,C 180,E1 12768.544,E2 12768.544} C_VEL
LIN {X 0,Y 324.573,Z 368.347,A -85,B 0,C 180,E1 12766.369,E2 12766.369} C_VEL
LIN {X 0,Y 327.714,Z 372.8,A -85,B 0,C 180,E1 12763.881,E2 12763.881} C_VEL
LIN {X 0,Y 330.187,Z 374.986,A -85,B 0,C 180,E1 12762.282,E2 12762.282} C_VEL
LIN {X 0,Y 334.021,Z 379.248,A -85,B 0,C 180,E1 12759.956,E2 12759.956} C_VEL
LIN {X 0,Y 338.1,Z 381.996,A -85,B 0,C 180,E1 12757.391,E2 12757.391} C_VEL
LIN {X 0,Y 341.965,Z 386.207,A -85,B 0,C 180,E1 12754.545,E2 12754.545} C_VEL
LIN {X 0,Y 345.212,Z 388.683,A -85,B 0,C 180,E1 12751.829,E2 12751.829} C_VEL
LIN {X 0,Y 347.469,Z 390.206,A -85,B 0,C 180,E1 12749.682,E2 12749.682} C_VEL
LIN {X 0,Y 349.798,Z 393.562,A -85,B 0,C 180,E1 12747.106,E2 12747.106} C_VEL
LIN {X 0,Y 352.945,Z 396.061,A -85,B 0,C 180,E1 12743.838,E2 12743.838} C_VEL
LIN {X 0,Y 354.587,Z 397.177,A -85,B 0,C 180,E1 12742.069,E2 12742.069} C_VEL
LIN {X 0,Y 356.993,Z 400.626,A -85,B 0,C 180,E1 12739.264,E2 12739.264} C_VEL
LIN {X 0,Y 360.106,Z 403.068,A -85,B 0,C 180,E1 12735.753,E2 12735.753} C_VEL
LIN {X 0,Y 361.925,Z 404.133,A -85,B 0,C 180,E1 12733.631,E2 12733.631} C_VEL
LIN {X 0,Y 364.1,Z 407.431,A -85,B 0,C 180,E1 12730.719,E2 12730.719} C_VEL
LIN {X 0,Y 366.533,Z 409.631,A -85,B 0,C 180,E1 12727.457,E2 12727.457} C_VEL
LIN {X 0,Y 369.081,Z 410.918,A -85,B 0,C 180,E1 12724.007,E2 12724.007} C_VEL
LIN {X 0,Y 370.831,Z 413.595,A -85,B 0,C 180,E1 12721.176,E2 12721.176} C_VEL
LIN {X 0,Y 372.788,Z 415.898,A -85,B 0,C 180,E1 12717.737,E2 12717.737} C_VEL
LIN {X 0,Y 374.613,Z 417.157,A -85,B 0,C 180,E1 12714.437,E2 12714.437} C_VEL
LIN {X 0,Y 376.477,Z 418.003,A -85,B 0,C 180,E1 12710.684,E2 12710.684} C_VEL
LIN {X 0,Y 377.522,Z 419.064,A -85,B 0,C 180,E1 12708.047,E2 12708.047} C_VEL
LIN {X 0,Y 378.562,Z 420.924,A -85,B 0,C 180,E1 12704.844,E2 12704.844} C_VEL
LIN {X 0,Y 379.523,Z 422.218,A -85,B 0,C 180,E1 12701.242,E2 12701.242} C_VEL
LIN {X 0,Y 380.152,Z 422.928,A -85,B 0,C 180,E1 12698.013,E2 12698.013} C_VEL
LIN {X 0,Y 380.699,Z 423.346,A -85,B 0,C 180,E1 12694.368,E2 12694.368} C_VEL
LIN {X 0,Y 380.854,Z 423.479,A -85,B 0,C 180,E1 12690.903,E2 12690.903} C_VEL
LIN {X 0,Y 380.809,Z 423.423,A -85,B 0,C 180,E1 12687.141,E2 12687.141} C_VEL
LIN {X 0,Y 380.433,Z 423.144,A -85,B 0,C 180,E1 12683.663,E2 12683.663} C_VEL
LIN {X 0,Y 379.76,Z 422.508,A -85,B 0,C 180,E1 12679.84,E2 12679.84} C_VEL
LIN {X 0,Y 378.922,Z 421.482,A -85,B 0,C 180,E1 12676.418,E2 12676.418} C_VEL
LIN {X 0,Y 377.814,Z 419.57,A -85,B 0,C 180,E1 12672.759,E2 12672.759} C_VEL
LIN {X 0,Y 376.836,Z 418.244,A -85,B 0,C 180,E1 12670.147,E2 12670.147} C_VEL
LIN {X 0,Y 375.172,Z 417.448,A -85,B 0,C 180,E1 12666.604,E2 12666.604} C_VEL
LIN {X 0,Y 373.11,Z 416.173,A -85,B 0,C 180,E1 12662.834,E2 12662.834} C_VEL
LIN {X 0,Y 371.158,Z 414.079,A -85,B 0,C 180,E1 12659.394,E2 12659.394} C_VEL
LIN {X 0,Y 369.157,Z 410.945,A -85,B 0,C 180,E1 12656.087,E2 12656.087} C_VEL
LIN {X 0,Y 366.68,Z 409.735,A -85,B 0,C 180,E1 12652.747,E2 12652.747} C_VEL
LIN {X 0,Y 364.256,Z 407.609,A -85,B 0,C 180,E1 12649.495,E2 12649.495} C_VEL
LIN {X 0,Y 362.027,Z 404.316,A -85,B 0,C 180,E1 12646.494,E2 12646.494} C_VEL
LIN {X 0,Y 360.876,Z 403.471,A -85,B 0,C 180,E1 12645.177,E2 12645.177} C_VEL
LIN {X 0,Y 358.012,Z 401.568,A -85,B 0,C 180,E1 12641.873,E2 12641.873} C_VEL
LIN {X 0,Y 355.508,Z 398.613,A -85,B 0,C 180,E1 12638.946,E2 12638.946} C_VEL
LIN {X 0,Y 354.1,Z 396.641,A -85,B 0,C 180,E1 12637.379,E2 12637.379} C_VEL
LIN {X 0,Y 351.006,Z 394.675,A -85,B 0,C 180,E1 12634.136,E2 12634.136} C_VEL
LIN {X 0,Y 348.193,Z 391.456,A -85,B 0,C 180,E1 12631.123,E2 12631.123} C_VEL
LIN {X 0,Y 347.027,Z 389.659,A -85,B 0,C 180,E1 12629.863,E2 12629.863} C_VEL
LIN {X 0,Y 343.825,Z 387.804,A -85,B 0,C 180,E1 12626.978,E2 12626.978} C_VEL
LIN {X 0,Y 340.391,Z 384.673,A -85,B 0,C 180,E1 12624.282,E2 12624.282} C_VEL
LIN {X 0,Y 338.1,Z 381.996,A -85,B 0,C 180,E1 12622.609,E2 12622.609} C_VEL
LIN {X 0,Y 334.021,Z 379.248,A -85,B 0,C 180,E1 12620.044,E2 12620.044} C_VEL
LIN {X 0,Y 330.187,Z 374.986,A -85,B 0,C 180,E1 12617.718,E2 12617.718} C_VEL
LIN {X 0,Y 325.663,Z 370.281,A -85,B 0,C 180,E1 12614.582,E2 12614.582} C_VEL
LIN {X 0,Y 324.283,Z 367.894,A -85,B 0,C 180,E1 12613.37,E2 12613.37} C_VEL
LIN {X 0,Y 320.934,Z 364.257,A -85,B 0,C 180,E1 12610.048,E2 12610.048} C_VEL
LIN {X 0,Y 319.935,Z 362.043,A -85,B 0,C 180,E1 12608.627,E2 12608.627} C_VEL
LIN {X 0,Y 316.841,Z 359.524,A -85,B 0,C 180,E1 12601.085,E2 12601.085} C_VEL
LIN {X 0,Y 317.206,Z 360.057,A -85,B 0,C 180,E1 12597.109,E2 12597.109} C_VEL
LIN {X 0,Y 320.104,Z 362.378,A -85,B 0,C 180,E1 12591.558,E2 12591.558} C_VEL
LIN {X 0,Y 322.252,Z 366.119,A -85,B 0,C 180,E1 12588.909,E2 12588.909} C_VEL
LIN {X 0,Y 322.518,Z 366.413,A -85,B 0,C 180,E1 12588.643,E2 12588.643} C_VEL
LIN {X 0,Y 323.175,Z 368.07,A -85,B 0,C 180,E1 12587.917,E2 12587.917} C_VEL
LIN {X 0,Y 323.97,Z 373.38,A -85,B 0,C 180,E1 12586.783,E2 12586.783} C_VEL
LIN {X 0,Y 324.818,Z 378.206,A -85,B 0,C 180,E1 12585.746,E2 12585.746} C_VEL
LIN {X 0,Y 325.518,Z 379.713,A -85,B 0,C 180,E1 12585.15,E2 12585.15} C_VEL
LIN {X 0,Y 327.441,Z 381.962,A -85,B 0,C 180,E1 12583.776,E2 12583.776} C_VEL
LIN {X 0,Y 331.358,Z 387.465,A -85,B 0,C 180,E1 12581.255,E2 12581.255} C_VEL
LIN {X 0,Y 335.342,Z 393.094,A -85,B 0,C 180,E1 12579.035,E2 12579.035} C_VEL
LIN {X 0,Y 339.991,Z 399.813,A -85,B 0,C 180,E1 12576.746,E2 12576.746} C_VEL
LIN {X 0,Y 346.081,Z 411.144,A -85,B 0,C 180,E1 12573.997,E2 12573.997} C_VEL
LIN {X 0,Y 351.656,Z 422.135,A -85,B 0,C 180,E1 12571.744,E2 12571.744} C_VEL
LIN {X 0,Y 352.915,Z 425.246,A -85,B 0,C 180,E1 12571.242,E2 12571.242} C_VEL
LIN {X 0,Y 340.544,Z 599.431,A -85,B 0,C 180,E1 12567.678,E2 12567.678} C_VEL
LIN {X 0,Y 337.325,Z 623.575,A -85,B 0,C 180,E1 12566.993,E2 12566.993} C_VEL
LIN {X 0,Y 333.847,Z 641.865,A -85,B 0,C 180,E1 12566.287,E2 12566.287} C_VEL
LIN {X 0,Y 329.607,Z 660.278,A -85,B 0,C 180,E1 12565.367,E2 12565.367} C_VEL
LIN {X 0,Y 323.452,Z 682.455,A -85,B 0,C 180,E1 12563.933,E2 12563.933} C_VEL
LIN {X 0,Y 317.951,Z 699.35,A -85,B 0,C 180,E1 12562.562,E2 12562.562} C_VEL
LIN {X 0,Y 312.133,Z 715.48,A -85,B 0,C 180,E1 12560.986,E2 12560.986} C_VEL
LIN {X 0,Y 304.451,Z 734.715,A -85,B 0,C 180,E1 12558.692,E2 12558.692} C_VEL
LIN {X 0,Y 297.586,Z 750.378,A -85,B 0,C 180,E1 12556.389,E2 12556.389} C_VEL
LIN {X 0,Y 291.084,Z 764.413,A -85,B 0,C 180,E1 12553.935,E2 12553.935} C_VEL
LIN {X 0,Y 283.252,Z 780.52,A -85,B 0,C 180,E1 12550.503,E2 12550.503} C_VEL
LIN {X 0,Y 277.492,Z 792.061,A -85,B 0,C 180,E1 12547.512,E2 12547.512} C_VEL
LIN {X 0,Y 272.132,Z 802.844,A -85,B 0,C 180,E1 12544.203,E2 12544.203} C_VEL
LIN {X 0,Y 266.349,Z 814.833,A -85,B 0,C 180,E1 12539.703,E2 12539.703} C_VEL
LIN {X 0,Y 262.509,Z 823.344,A -85,B 0,C 180,E1 12535.734,E2 12535.734} C_VEL
LIN {X 0,Y 259.665,Z 830.475,A -85,B 0,C 180,E1 12531.694,E2 12531.694} C_VEL
LIN {X 0,Y 257.344,Z 837.613,A -85,B 0,C 180,E1 12526.476,E2 12526.476} C_VEL
LIN {X 0,Y 256.4,Z 841.76,A -85,B 0,C 180,E1 12522.385,E2 12522.385} C_VEL
LIN {X 0,Y 256.041,Z 844.595,A -85,B 0,C 180,E1 12518.534,E2 12518.534} C_VEL
LIN {X 0,Y 255.966,Z 846.393,A -85,B 0,C 180,E1 12514.705,E2 12514.705} C_VEL
LIN {X 0,Y 255.982,Z 847.218,A -85,B 0,C 180,E1 12510.448,E2 12510.448} C_VEL
LIN {X 0,Y 255.964,Z 846.642,A -85,B 0,C 180,E1 12505.968,E2 12505.968} C_VEL
LIN {X 0,Y 256.031,Z 844.734,A -85,B 0,C 180,E1 12501.692,E2 12501.692} C_VEL
LIN {X 0,Y 256.366,Z 841.955,A -85,B 0,C 180,E1 12497.842,E2 12497.842} C_VEL
LIN {X 0,Y 257.274,Z 837.866,A -85,B 0,C 180,E1 12493.751,E2 12493.751} C_VEL
LIN {X 0,Y 259.411,Z 831.218,A -85,B 0,C 180,E1 12488.759,E2 12488.759} C_VEL
LIN {X 0,Y 262.326,Z 823.778,A -85,B 0,C 180,E1 12484.489,E2 12484.489} C_VEL
LIN {X 0,Y 265.867,Z 815.832,A -85,B 0,C 180,E1 12480.733,E2 12480.733} C_VEL
LIN {X 0,Y 271.239,Z 804.73,A -85,B 0,C 180,E1 12476.418,E2 12476.418} C_VEL
LIN {X 0,Y 277.133,Z 792.78,A -85,B 0,C 180,E1 12472.692,E2 12472.692} C_VEL
LIN {X 0,Y 282.846,Z 781.323,A -85,B 0,C 180,E1 12469.693,E2 12469.693} C_VEL
LIN {X 0,Y 290.168,Z 766.403,A -85,B 0,C 180,E1 12466.438,E2 12466.438} C_VEL
LIN {X 0,Y 297.085,Z 751.484,A -85,B 0,C 180,E1 12463.789,E2 12463.789} C_VEL
LIN {X 0,Y 303.522,Z 736.851,A -85,B 0,C 180,E1 12461.603,E2 12461.603} C_VEL
LIN {X 0,Y 310.969,Z 718.669,A -85,B 0,C 180,E1 12459.353,E2 12459.353} C_VEL
LIN {X 0,Y 317.357,Z 701.088,A -85,B 0,C 180,E1 12457.594,E2 12457.594} C_VEL
LIN {X 0,Y 322.833,Z 684.429,A -85,B 0,C 180,E1 12456.217,E2 12456.217} C_VEL
LIN {X 0,Y 328.588,Z 664.511,A -85,B 0,C 180,E1 12454.87,E2 12454.87} C_VEL
LIN {X 0,Y 333.358,Z 644.214,A -85,B 0,C 180,E1 12453.819,E2 12453.819} C_VEL
LIN {X 0,Y 336.897,Z 626.023,A -85,B 0,C 180,E1 12453.094,E2 12453.094} C_VEL
LIN {X 0,Y 340.129,Z 603.941,A -85,B 0,C 180,E1 12452.428,E2 12452.428} C_VEL
LIN {X 0,Y 343.194,Z 563.726,A -85,B 0,C 180,E1 12451.564,E2 12451.564} C_VEL
LIN {X 0,Y 352.875,Z 424.743,A -85,B 0,C 180,E1 12448.726,E2 12448.726} C_VEL
LIN {X 0,Y 347.467,Z 413.752,A -85,B 0,C 180,E1 12446.581,E2 12446.581} C_VEL
LIN {X 0,Y 341.986,Z 403.457,A -85,B 0,C 180,E1 12444.194,E2 12444.194} C_VEL
LIN {X 0,Y 338.973,Z 398.349,A -85,B 0,C 180,E1 12442.777,E2 12442.777} C_VEL
LIN {X 0,Y 333.68,Z 390.616,A -85,B 0,C 180,E1 12440.065,E2 12440.065} C_VEL
LIN {X 0,Y 329.722,Z 385.201,A -85,B 0,C 180,E1 12437.744,E2 12437.744} C_VEL
LIN {X 0,Y 326.48,Z 380.707,A -85,B 0,C 180,E1 12435.544,E2 12435.544} C_VEL
LIN {X 0,Y 323.354,Z 376.436,A -85,B 0,C 180,E1 12433.046,E2 12433.046} C_VEL
LIN {X 0,Y 322.584,Z 375.405,A -85,B 0,C 180,E1 12432.349,E2 12432.349} C_VEL
LIN {X 0,Y 319.459,Z 371.535,A -85,B 0,C 180,E1 12429.003,E2 12429.003} C_VEL
LIN {X 0,Y 318.749,Z 369.916,A -85,B 0,C 180,E1 12427.933,E2 12427.933} C_VEL
LIN {X 0,Y 315.859,Z 367.451,A -85,B 0,C 180,E1 12420.544,E2 12420.544} C_VEL
LIN {X 0,Y 316.309,Z 368.112,A -85,B 0,C 180,E1 12416.375,E2 12416.375} C_VEL
LIN {X 0,Y 318.94,Z 370.24,A -85,B 0,C 180,E1 12411.345,E2 12411.345} C_VEL
LIN {X 0,Y 321.038,Z 373.929,A -85,B 0,C 180,E1 12408.685,E2 12408.685} C_VEL
LIN {X 0,Y 323.191,Z 376.086,A -85,B 0,C 180,E1 12406.675,E2 12406.675} C_VEL
LIN {X 0,Y 326.384,Z 380.608,A -85,B 0,C 180,E1 12404.087,E2 12404.087} C_VEL
LIN {X 0,Y 328.685,Z 382.722,A -85,B 0,C 180,E1 12402.564,E2 12402.564} C_VEL
LIN {X 0,Y 332.648,Z 387.06,A -85,B 0,C 180,E1 12400.145,E2 12400.145} C_VEL
LIN {X 0,Y 336.917,Z 389.886,A -85,B 0,C 180,E1 12397.491,E2 12397.491} C_VEL
LIN {X 0,Y 340.225,Z 393.63,A -85,B 0,C 180,E1 12395.057,E2 12395.057} C_VEL
LIN {X 0,Y 343.526,Z 396.242,A -85,B 0,C 180,E1 12392.433,E2 12392.433} C_VEL
LIN {X 0,Y 346.223,Z 397.973,A -85,B 0,C 180,E1 12389.931,E2 12389.931} C_VEL
LIN {X 0,Y 348.548,Z 401.323,A -85,B 0,C 180,E1 12387.364,E2 12387.364} C_VEL
LIN {X 0,Y 351.672,Z 403.867,A -85,B 0,C 180,E1 12384.123,E2 12384.123} C_VEL
LIN {X 0,Y 353.437,Z 405.06,A -85,B 0,C 180,E1 12382.232,E2 12382.232} C_VEL
LIN {X 0,Y 355.765,Z 408.394,A -85,B 0,C 180,E1 12379.518,E2 12379.518} C_VEL
LIN {X 0,Y 358.831,Z 410.868,A -85,B 0,C 180,E1 12376.067,E2 12376.067} C_VEL
LIN {X 0,Y 360.792,Z 412.021,A -85,B 0,C 180,E1 12373.787,E2 12373.787} C_VEL
LIN {X 0,Y 362.937,Z 415.214,A -85,B 0,C 180,E1 12370.969,E2 12370.969} C_VEL
LIN {X 0,Y 365.511,Z 417.562,A -85,B 0,C 180,E1 12367.505,E2 12367.505} C_VEL
LIN {X 0,Y 367.922,Z 418.801,A -85,B 0,C 180,E1 12364.23,E2 12364.23} C_VEL
LIN {X 0,Y 368.713,Z 419.815,A -85,B 0,C 180,E1 12363.028,E2 12363.028} C_VEL
LIN {X 0,Y 370.519,Z 422.559,A -85,B 0,C 180,E1 12359.948,E2 12359.948} C_VEL
LIN {X 0,Y 372.46,Z 424.334,A -85,B 0,C 180,E1 12356.629,E2 12356.629} C_VEL
LIN {X 0,Y 374.422,Z 425.512,A -85,B 0,C 180,E1 12352.885,E2 12352.885} C_VEL
LIN {X 0,Y 375.987,Z 426.3,A -85,B 0,C 180,E1 12349.576,E2 12349.576} C_VEL
LIN {X 0,Y 377.184,Z 428.245,A -85,B 0,C 180,E1 12346.161,E2 12346.161} C_VEL
LIN {X 0,Y 378.087,Z 429.612,A -85,B 0,C 180,E1 12342.99,E2 12342.99} C_VEL
LIN {X 0,Y 378.988,Z 430.604,A -85,B 0,C 180,E1 12339.414,E2 12339.414} C_VEL
LIN {X 0,Y 379.498,Z 431.161,A -85,B 0,C 180,E1 12335.898,E2 12335.898} C_VEL
LIN {X 0,Y 379.89,Z 431.416,A -85,B 0,C 180,E1 12332.263,E2 12332.263} C_VEL
LIN {X 0,Y 379.864,Z 431.416,A -85,B 0,C 180,E1 12328.793,E2 12328.793} C_VEL
LIN {X 0,Y 379.685,Z 431.233,A -85,B 0,C 180,E1 12325.166,E2 12325.166} C_VEL
LIN {X 0,Y 379.114,Z 430.796,A -85,B 0,C 180,E1 12321.66,E2 12321.66} C_VEL
LIN {X 0,Y 378.414,Z 430.02,A -85,B 0,C 180,E1 12318.107,E2 12318.107} C_VEL
LIN {X 0,Y 377.404,Z 428.608,A -85,B 0,C 180,E1 12314.638,E2 12314.638} C_VEL
LIN {X 0,Y 376.381,Z 426.727,A -85,B 0,C 180,E1 12311.411,E2 12311.411} C_VEL
LIN {X 0,Y 375.028,Z 425.74,A -85,B 0,C 180,E1 12308.249,E2 12308.249} C_VEL
LIN {X 0,Y 373.194,Z 424.88,A -85,B 0,C 180,E1 12304.787,E2 12304.787} C_VEL
LIN {X 0,Y 371.179,Z 423.2,A -85,B 0,C 180,E1 12301.1,E2 12301.1} C_VEL
LIN {X 0,Y 369.269,Z 420.78,A -85,B 0,C 180,E1 12297.941,E2 12297.941} C_VEL
LIN {X 0,Y 368.063,Z 418.849,A -85,B 0,C 180,E1 12295.949,E2 12295.949} C_VEL
LIN {X 0,Y 365.599,Z 417.624,A -85,B 0,C 180,E1 12292.618,E2 12292.618} C_VEL
LIN {X 0,Y 363.098,Z 415.408,A -85,B 0,C 180,E1 12289.262,E2 12289.262} C_VEL
LIN {X 0,Y 360.873,Z 412.168,A -85,B 0,C 180,E1 12286.314,E2 12286.314} C_VEL
LIN {X 0,Y 358.943,Z 410.93,A -85,B 0,C 180,E1 12284.057,E2 12284.057} C_VEL
LIN {X 0,Y 355.935,Z 408.569,A -85,B 0,C 180,E1 12280.671,E2 12280.671} C_VEL
LIN {X 0,Y 353.673,Z 405.464,A -85,B 0,C 180,E1 12278.046,E2 12278.046} C_VEL
LIN {X 0,Y 352.88,Z 404.469,A -85,B 0,C 180,E1 12277.122,E2 12277.122} C_VEL
LIN {X 0,Y 349.762,Z 402.449,A -85,B 0,C 180,E1 12273.879,E2 12273.879} C_VEL
LIN {X 0,Y 346.947,Z 399.198,A -85,B 0,C 180,E1 12270.862,E2 12270.862} C_VEL
LIN {X 0,Y 345.8,Z 397.503,A -85,B 0,C 180,E1 12269.632,E2 12269.632} C_VEL
LIN {X 0,Y 342.436,Z 395.537,A -85,B 0,C 180,E1 12266.69,E2 12266.69} C_VEL
LIN {X 0,Y 338.915,Z 392.269,A -85,B 0,C 180,E1 12263.932,E2 12263.932} C_VEL
LIN {X 0,Y 336.668,Z 389.757,A -85,B 0,C 180,E1 12262.342,E2 12262.342} C_VEL
LIN {X 0,Y 332.247,Z 386.729,A -85,B 0,C 180,E1 12259.625,E2 12259.625} C_VEL
LIN {X 0,Y 327.78,Z 381.756,A -85,B 0,C 180,E1 12256.845,E2 12256.845} C_VEL
LIN {X 0,Y 324.256,Z 377.984,A -85,B 0,C 180,E1 12254.281,E2 12254.281} C_VEL
LIN {X 0,Y 322.704,Z 375.488,A -85,B 0,C 180,E1 12252.89,E2 12252.89} C_VEL
LIN {X 0,Y 319.537,Z 371.684,A -85,B 0,C 180,E1 12249.546,E2 12249.546} C_VEL
LIN {X 0,Y 318.696,Z 369.879,A -85,B 0,C 180,E1 12248.298,E2 12248.298} C_VEL
LIN {X 0,Y 315.866,Z 367.467,A -85,B 0,C 180,E1 12241.088,E2 12241.088} C_VEL
LIN {X 0,Y 316.23,Z 368.014,A -85,B 0,C 180,E1 12237.1,E2 12237.1} C_VEL
LIN {X 0,Y 318.927,Z 370.234,A -85,B 0,C 180,E1 12231.799,E2 12231.799} C_VEL
LIN {X 0,Y 321.106,Z 374.015,A -85,B 0,C 180,E1 12229.051,E2 12229.051} C_VEL
LIN {X 0,Y 323.17,Z 376.072,A -85,B 0,C 180,E1 12227.129,E2 12227.129} C_VEL
LIN {X 0,Y 325.518,Z 379.713,A -85,B 0,C 180,E1 12225.15,E2 12225.15} C_VEL
LIN {X 0,Y 327.085,Z 382.73,A -85,B 0,C 180,E1 12223.929,E2 12223.929} C_VEL
LIN {X 0,Y 329.194,Z 389.856,A -85,B 0,C 180,E1 12222.217,E2 12222.217} C_VEL
LIN {X 0,Y 331.57,Z 397.19,A -85,B 0,C 180,E1 12220.527,E2 12220.527} C_VEL
LIN {X 0,Y 332.391,Z 398.815,A -85,B 0,C 180,E1 12220.035,E2 12220.035} C_VEL
LIN {X 0,Y 337.717,Z 406.862,A -85,B 0,C 180,E1 12217.272,E2 12217.272} C_VEL
LIN {X 0,Y 343.476,Z 417.889,A -85,B 0,C 180,E1 12214.572,E2 12214.572} C_VEL
LIN {X 0,Y 348.721,Z 428.556,A -85,B 0,C 180,E1 12212.368,E2 12212.368} C_VEL
LIN {X 0,Y 348.65,Z 431.283,A -85,B 0,C 180,E1 12212.272,E2 12212.272} C_VEL
LIN {X 0,Y 336.322,Z 599.137,A -85,B 0,C 180,E1 12208.836,E2 12208.836} C_VEL
LIN {X 0,Y 333.012,Z 623.325,A -85,B 0,C 180,E1 12208.154,E2 12208.154} C_VEL
LIN {X 0,Y 329.274,Z 642.398,A -85,B 0,C 180,E1 12207.418,E2 12207.418} C_VEL
LIN {X 0,Y 324.691,Z 661.607,A -85,B 0,C 180,E1 12206.452,E2 12206.452} C_VEL
LIN {X 0,Y 318.425,Z 683.19,A -85,B 0,C 180,E1 12205.037,E2 12205.037} C_VEL
LIN {X 0,Y 312.764,Z 699.967,A -85,B 0,C 180,E1 12203.667,E2 12203.667} C_VEL
LIN {X 0,Y 306.143,Z 717.644,A -85,B 0,C 180,E1 12201.913,E2 12201.913} C_VEL
LIN {X 0,Y 298.416,Z 735.98,A -85,B 0,C 180,E1 12199.661,E2 12199.661} C_VEL
LIN {X 0,Y 291.715,Z 750.676,A -85,B 0,C 180,E1 12197.468,E2 12197.468} C_VEL
LIN {X 0,Y 284.726,Z 765.152,A -85,B 0,C 180,E1 12194.896,E2 12194.896} C_VEL
LIN {X 0,Y 277.011,Z 780.263,A -85,B 0,C 180,E1 12191.615,E2 12191.615} C_VEL
LIN {X 0,Y 270.788,Z 792.136,A -85,B 0,C 180,E1 12188.484,E2 12188.484} C_VEL
LIN {X 0,Y 264.988,Z 803.227,A -85,B 0,C 180,E1 12184.996,E2 12184.996} C_VEL
LIN {X 0,Y 258.922,Z 815.075,A -85,B 0,C 180,E1 12180.388,E2 12180.388} C_VEL
LIN {X 0,Y 255.079,Z 823.087,A -85,B 0,C 180,E1 12176.541,E2 12176.541} C_VEL
LIN {X 0,Y 251.879,Z 830.59,A -85,B 0,C 180,E1 12172.154,E2 12172.154} C_VEL
LIN {X 0,Y 249.499,Z 837.359,A -85,B 0,C 180,E1 12167.01,E2 12167.01} C_VEL
LIN {X 0,Y 248.459,Z 841.507,A -85,B 0,C 180,E1 12162.787,E2 12162.787} C_VEL
LIN {X 0,Y 248.049,Z 844.344,A -85,B 0,C 180,E1 12158.811,E2 12158.811} C_VEL
LIN {X 0,Y 247.968,Z 846.143,A -85,B 0,C 180,E1 12154.857,E2 12154.857} C_VEL
LIN {X 0,Y 247.986,Z 846.943,A -85,B 0,C 180,E1 12150.693,E2 12150.693} C_VEL
LIN {X 0,Y 247.966,Z 846.475,A -85,B 0,C 180,E1 12146.07,E2 12146.07} C_VEL
LIN {X 0,Y 248.033,Z 844.623,A -85,B 0,C 180,E1 12141.656,E2 12141.656} C_VEL
LIN {X 0,Y 248.421,Z 841.703,A -85,B 0,C 180,E1 12137.447,E2 12137.447} C_VEL
LIN {X 0,Y 249.421,Z 837.612,A -85,B 0,C 180,E1 12133.225,E2 12133.225} C_VEL
LIN {X 0,Y 251.743,Z 830.962,A -85,B 0,C 180,E1 12128.079,E2 12128.079} C_VEL
LIN {X 0,Y 254.882,Z 823.521,A -85,B 0,C 180,E1 12123.688,E2 12123.688} C_VEL
LIN {X 0,Y 258.669,Z 815.574,A -85,B 0,C 180,E1 12119.835,E2 12119.835} C_VEL
LIN {X 0,Y 264.351,Z 804.509,A -85,B 0,C 180,E1 12115.436,E2 12115.436} C_VEL
LIN {X 0,Y 270.586,Z 792.522,A -85,B 0,C 180,E1 12111.628,E2 12111.628} C_VEL
LIN {X 0,Y 276.585,Z 781.066,A -85,B 0,C 180,E1 12108.583,E2 12108.583} C_VEL
LIN {X 0,Y 284.318,Z 766.001,A -85,B 0,C 180,E1 12105.265,E2 12105.265} C_VEL
LIN {X 0,Y 291.369,Z 751.414,A -85,B 0,C 180,E1 12102.652,E2 12102.652} C_VEL
LIN {X 0,Y 297.95,Z 737.018,A -85,B 0,C 180,E1 12100.483,E2 12100.483} C_VEL
LIN {X 0,Y 305.564,Z 719.184,A -85,B 0,C 180,E1 12098.252,E2 12098.252} C_VEL
LIN {X 0,Y 312.396,Z 701.011,A -85,B 0,C 180,E1 12096.428,E2 12096.428} C_VEL
LIN {X 0,Y 318.106,Z 684.177,A -85,B 0,C 180,E1 12095.038,E2 12095.038} C_VEL
LIN {X 0,Y 323.943,Z 664.592,A -85,B 0,C 180,E1 12093.716,E2 12093.716} C_VEL
LIN {X 0,Y 328.939,Z 643.964,A -85,B 0,C 180,E1 12092.652,E2 12092.652} C_VEL
LIN {X 0,Y 332.605,Z 625.597,A -85,B 0,C 180,E1 12091.927,E2 12091.927} C_VEL
LIN {X 0,Y 335.918,Z 603.382,A -85,B 0,C 180,E1 12091.264,E2 12091.264} C_VEL
LIN {X 0,Y 339.13,Z 562.456,A -85,B 0,C 180,E1 12090.387,E2 12090.387} C_VEL
LIN {X 0,Y 348.767,Z 428.659,A -85,B 0,C 180,E1 12087.651,E2 12087.651} C_VEL
LIN {X 0,Y 343.565,Z 418.066,A -85,B 0,C 180,E1 12085.467,E2 12085.467} C_VEL
LIN {X 0,Y 338.441,Z 408.274,A -85,B 0,C 180,E1 12083.09,E2 12083.09} C_VEL
LIN {X 0,Y 334.981,Z 402.612,A -85,B 0,C 180,E1 12081.355,E2 12081.355} C_VEL
LIN {X 0,Y 330.637,Z 396.482,A -85,B 0,C 180,E1 12078.971,E2 12078.971} C_VEL
LIN {X 0,Y 327.944,Z 392.584,A -85,B 0,C 180,E1 12077.293,E2 12077.293} C_VEL
LIN {X 0,Y 324.912,Z 388.281,A -85,B 0,C 180,E1 12075.163,E2 12075.163} C_VEL
LIN {X 0,Y 321.796,Z 383.8,A -85,B 0,C 180,E1 12072.562,E2 12072.562} C_VEL
LIN {X 0,Y 318.151,Z 379.087,A -85,B 0,C 180,E1 12068.585,E2 12068.585} C_VEL
LIN {X 0,Y 317.519,Z 377.747,A -85,B 0,C 180,E1 12067.6,E2 12067.6} C_VEL
LIN {X 0,Y 314.884,Z 375.394,A -85,B 0,C 180,E1 12060.546,E2 12060.546} C_VEL
LIN {X 0,Y 315.285,Z 376.005,A -85,B 0,C 180,E1 12056.542,E2 12056.542} C_VEL
LIN {X 0,Y 317.769,Z 378.092,A -85,B 0,C 180,E1 12051.587,E2 12051.587} C_VEL
LIN {X 0,Y 320.065,Z 382.015,A -85,B 0,C 180,E1 12048.65,E2 12048.65} C_VEL
LIN {X 0,Y 321.907,Z 383.999,A -85,B 0,C 180,E1 12046.895,E2 12046.895} C_VEL
LIN {X 0,Y 325.179,Z 388.53,A -85,B 0,C 180,E1 12044.21,E2 12044.21} C_VEL
LIN {X 0,Y 327.191,Z 390.453,A -85,B 0,C 180,E1 12042.849,E2 12042.849} C_VEL
LIN {X 0,Y 331.268,Z 394.869,A -85,B 0,C 180,E1 12040.335,E2 12040.335} C_VEL
LIN {X 0,Y 336.072,Z 398.301,A -85,B 0,C 180,E1 12037.339,E2 12037.339} C_VEL
LIN {X 0,Y 339.175,Z 401.664,A -85,B 0,C 180,E1 12035.068,E2 12035.068} C_VEL
LIN {X 0,Y 342.609,Z 404.266,A -85,B 0,C 180,E1 12032.353,E2 12032.353} C_VEL
LIN {X 0,Y 345.047,Z 405.861,A -85,B 0,C 180,E1 12030.105,E2 12030.105} C_VEL
LIN {X 0,Y 347.305,Z 409.081,A -85,B 0,C 180,E1 12027.624,E2 12027.624} C_VEL
LIN {X 0,Y 350.394,Z 411.671,A -85,B 0,C 180,E1 12024.4,E2 12024.4} C_VEL
LIN {X 0,Y 352.291,Z 412.94,A -85,B 0,C 180,E1 12022.396,E2 12022.396} C_VEL
LIN {X 0,Y 354.543,Z 416.161,A -85,B 0,C 180,E1 12019.774,E2 12019.774} C_VEL
LIN {X 0,Y 357.616,Z 418.694,A -85,B 0,C 180,E1 12016.324,E2 12016.324} C_VEL
LIN {X 0,Y 359.731,Z 420.034,A -85,B 0,C 180,E1 12013.856,E2 12013.856} C_VEL
LIN {X 0,Y 362.049,Z 423.328,A -85,B 0,C 180,E1 12010.826,E2 12010.826} C_VEL
LIN {X 0,Y 364.519,Z 425.515,A -85,B 0,C 180,E1 12007.511,E2 12007.511} C_VEL
LIN {X 0,Y 367.01,Z 426.767,A -85,B 0,C 180,E1 12004.139,E2 12004.139} C_VEL
LIN {X 0,Y 369.274,Z 430.198,A -85,B 0,C 180,E1 12000.419,E2 12000.419} C_VEL
LIN {X 0,Y 371.195,Z 432.107,A -85,B 0,C 180,E1 11997.078,E2 11997.078} C_VEL
LIN {X 0,Y 373.277,Z 433.372,A -85,B 0,C 180,E1 11993.255,E2 11993.255} C_VEL
LIN {X 0,Y 374.896,Z 434.166,A -85,B 0,C 180,E1 11989.798,E2 11989.798} C_VEL
LIN {X 0,Y 376.019,Z 435.838,A -85,B 0,C 180,E1 11986.812,E2 11986.812} C_VEL
LIN {X 0,Y 377.016,Z 437.445,A -85,B 0,C 180,E1 11983.339,E2 11983.339} C_VEL
LIN {X 0,Y 377.877,Z 438.465,A -85,B 0,C 180,E1 11979.903,E2 11979.903} C_VEL
LIN {X 0,Y 378.485,Z 439.052,A -85,B 0,C 180,E1 11976.218,E2 11976.218} C_VEL
LIN {X 0,Y 378.873,Z 439.315,A -85,B 0,C 180,E1 11972.723,E2 11972.723} C_VEL
LIN {X 0,Y 378.899,Z 439.36,A -85,B 0,C 180,E1 11969.093,E2 11969.093} C_VEL
LIN {X 0,Y 378.742,Z 439.225,A -85,B 0,C 180,E1 11965.609,E2 11965.609} C_VEL
LIN {X 0,Y 378.189,Z 438.804,A -85,B 0,C 180,E1 11961.945,E2 11961.945} C_VEL
LIN {X 0,Y 377.532,Z 438.063,A -85,B 0,C 180,E1 11958.543,E2 11958.543} C_VEL
LIN {X 0,Y 376.513,Z 436.717,A -85,B 0,C 180,E1 11954.916,E2 11954.916} C_VEL
LIN {X 0,Y 375.541,Z 434.952,A -85,B 0,C 180,E1 11951.895,E2 11951.895} C_VEL
LIN {X 0,Y 374.454,Z 433.861,A -85,B 0,C 180,E1 11949.157,E2 11949.157} C_VEL
LIN {X 0,Y 372.563,Z 433.005,A -85,B 0,C 180,E1 11945.42,E2 11945.42} C_VEL
LIN {X 0,Y 370.781,Z 431.777,A -85,B 0,C 180,E1 11942.189,E2 11942.189} C_VEL
LIN {X 0,Y 368.734,Z 429.42,A -85,B 0,C 180,E1 11938.627,E2 11938.627} C_VEL
LIN {X 0,Y 367.01,Z 426.767,A -85,B 0,C 180,E1 11935.861,E2 11935.861} C_VEL
LIN {X 0,Y 364.519,Z 425.514,A -85,B 0,C 180,E1 11932.489,E2 11932.489} C_VEL
LIN {X 0,Y 361.894,Z 423.148,A -85,B 0,C 180,E1 11928.96,E2 11928.96} C_VEL
LIN {X 0,Y 359.589,Z 419.772,A -85,B 0,C 180,E1 11925.963,E2 11925.963} C_VEL
LIN {X 0,Y 356.538,Z 417.965,A -85,B 0,C 180,E1 11922.479,E2 11922.479} C_VEL
LIN {X 0,Y 353.619,Z 414.947,A -85,B 0,C 180,E1 11919.089,E2 11919.089} C_VEL
LIN {X 0,Y 351.782,Z 412.363,A -85,B 0,C 180,E1 11916.998,E2 11916.998} C_VEL
LIN {X 0,Y 348.525,Z 410.222,A -85,B 0,C 180,E1 11913.62,E2 11913.62} C_VEL
LIN {X 0,Y 345.692,Z 406.94,A -85,B 0,C 180,E1 11910.601,E2 11910.601} C_VEL
LIN {X 0,Y 344.519,Z 405.324,A -85,B 0,C 180,E1 11909.371,E2 11909.371} C_VEL
LIN {X 0,Y 341.125,Z 403.317,A -85,B 0,C 180,E1 11906.457,E2 11906.457} C_VEL
LIN {X 0,Y 337.511,Z 399.988,A -85,B 0,C 180,E1 11903.666,E2 11903.666} C_VEL
LIN {X 0,Y 335.232,Z 397.514,A -85,B 0,C 180,E1 11902.074,E2 11902.074} C_VEL
LIN {X 0,Y 330.7,Z 394.397,A -85,B 0,C 180,E1 11899.334,E2 11899.334} C_VEL
LIN {X 0,Y 326.306,Z 389.461,A -85,B 0,C 180,E1 11896.557,E2 11896.557} C_VEL
LIN {X 0,Y 322.858,Z 385.685,A -85,B 0,C 180,E1 11893.978,E2 11893.978} C_VEL
LIN {X 0,Y 321.345,Z 383.218,A -85,B 0,C 180,E1 11892.58,E2 11892.58} C_VEL
LIN {X 0,Y 318.287,Z 379.373,A -85,B 0,C 180,E1 11889.219,E2 11889.219} C_VEL
LIN {X 0,Y 317.598,Z 377.774,A -85,B 0,C 180,E1 11888.144,E2 11888.144} C_VEL
LIN {X 0,Y 314.878,Z 375.402,A -85,B 0,C 180,E1 11880.91,E2 11880.91} C_VEL
LIN {X 0,Y 315.303,Z 376.036,A -85,B 0,C 180,E1 11876.91,E2 11876.91} C_VEL
LIN {X 0,Y 317.756,Z 378.082,A -85,B 0,C 180,E1 11872.042,E2 11872.042} C_VEL
LIN {X 0,Y 320.131,Z 382.101,A -85,B 0,C 180,E1 11869.017,E2 11869.017} C_VEL
LIN {X 0,Y 321.796,Z 383.805,A -85,B 0,C 180,E1 11867.438,E2 11867.438} C_VEL
LIN {X 0,Y 324.912,Z 388.284,A -85,B 0,C 180,E1 11864.837,E2 11864.837} C_VEL
LIN {X 0,Y 329.537,Z 394.828,A -85,B 0,C 180,E1 11861.698,E2 11861.698} C_VEL
LIN {X 0,Y 332.391,Z 398.815,A -85,B 0,C 180,E1 11860.035,E2 11860.035} C_VEL
LIN {X 0,Y 334.203,Z 403.052,A -85,B 0,C 180,E1 11858.959,E2 11858.959} C_VEL
LIN {X 0,Y 336.737,Z 412.422,A -85,B 0,C 180,E1 11857.368,E2 11857.368} C_VEL
LIN {X 0,Y 339.302,Z 421.069,A -85,B 0,C 180,E1 11855.921,E2 11855.921} C_VEL
LIN {X 0,Y 339.881,Z 422.451,A -85,B 0,C 180,E1 11855.637,E2 11855.637} C_VEL
LIN {X 0,Y 344.84,Z 432.911,A -85,B 0,C 180,E1 11853.417,E2 11853.417} C_VEL
LIN {X 0,Y 332.218,Z 599.077,A -85,B 0,C 180,E1 11850.018,E2 11850.018} C_VEL
LIN {X 0,Y 328.712,Z 623.769,A -85,B 0,C 180,E1 11849.32,E2 11849.32} C_VEL
LIN {X 0,Y 325.006,Z 642.148,A -85,B 0,C 180,E1 11848.615,E2 11848.615} C_VEL
LIN {X 0,Y 320.196,Z 661.754,A -85,B 0,C 180,E1 11847.635,E2 11847.635} C_VEL
LIN {X 0,Y 313.846,Z 682.938,A -85,B 0,C 180,E1 11846.251,E2 11846.251} C_VEL
LIN {X 0,Y 308.014,Z 699.714,A -85,B 0,C 180,E1 11844.886,E2 11844.886} C_VEL
LIN {X 0,Y 301.174,Z 717.391,A -85,B 0,C 180,E1 11843.136,E2 11843.136} C_VEL
LIN {X 0,Y 293.165,Z 735.747,A -85,B 0,C 180,E1 11840.88,E2 11840.88} C_VEL
LIN {X 0,Y 286.219,Z 750.42,A -85,B 0,C 180,E1 11838.681,E2 11838.681} C_VEL
LIN {X 0,Y 278.698,Z 765.393,A -85,B 0,C 180,E1 11835.996,E2 11835.996} C_VEL
LIN {X 0,Y 270.435,Z 780.809,A -85,B 0,C 180,E1 11832.576,E2 11832.576} C_VEL
LIN {X 0,Y 263.982,Z 792.547,A -85,B 0,C 180,E1 11829.406,E2 11829.406} C_VEL
LIN {X 0,Y 257.231,Z 804.881,A -85,B 0,C 180,E1 11825.391,E2 11825.391} C_VEL
LIN {X 0,Y 251.534,Z 815.317,A -85,B 0,C 180,E1 11821.114,E2 11821.114} C_VEL
LIN {X 0,Y 247.489,Z 823.264,A -85,B 0,C 180,E1 11817.162,E2 11817.162} C_VEL
LIN {X 0,Y 243.965,Z 831.077,A -85,B 0,C 180,E1 11812.404,E2 11812.404} C_VEL
LIN {X 0,Y 241.587,Z 837.357,A -85,B 0,C 180,E1 11807.336,E2 11807.336} C_VEL
LIN {X 0,Y 240.485,Z 841.45,A -85,B 0,C 180,E1 11802.974,E2 11802.974} C_VEL
LIN {X 0,Y 240.044,Z 844.372,A -85,B 0,C 180,E1 11798.624,E2 11798.624} C_VEL
LIN {X 0,Y 239.969,Z 846.307,A -85,B 0,C 180,E1 11793.822,E2 11793.822} C_VEL
LIN {X 0,Y 239.99,Z 846.682,A -85,B 0,C 180,E1 11789.179,E2 11789.179} C_VEL
LIN {X 0,Y 239.97,Z 845.894,A -85,B 0,C 180,E1 11784.98,E2 11784.98} C_VEL
LIN {X 0,Y 240.062,Z 844.093,A -85,B 0,C 180,E1 11780.894,E2 11780.894} C_VEL
LIN {X 0,Y 240.528,Z 841.254,A -85,B 0,C 180,E1 11776.784,E2 11776.784} C_VEL
LIN {X 0,Y 241.76,Z 836.851,A -85,B 0,C 180,E1 11772.179,E2 11772.179} C_VEL
LIN {X 0,Y 244.409,Z 829.962,A -85,B 0,C 180,E1 11766.876,E2 11766.876} C_VEL
LIN {X 0,Y 247.7,Z 822.83,A -85,B 0,C 180,E1 11762.603,E2 11762.603} C_VEL
LIN {X 0,Y 252.078,Z 814.318,A -85,B 0,C 180,E1 11758.429,E2 11758.429} C_VEL
LIN {X 0,Y 258.58,Z 802.328,A -85,B 0,C 180,E1 11753.73,E2 11753.73} C_VEL
LIN {X 0,Y 264.531,Z 791.546,A -85,B 0,C 180,E1 11750.301,E2 11750.301} C_VEL
LIN {X 0,Y 271.336,Z 779.203,A -85,B 0,C 180,E1 11747.024,E2 11747.024} C_VEL
LIN {X 0,Y 279.687,Z 763.417,A -85,B 0,C 180,E1 11743.627,E2 11743.627} C_VEL
LIN {X 0,Y 286.488,Z 749.867,A -85,B 0,C 180,E1 11741.229,E2 11741.229} C_VEL
LIN {X 0,Y 293.752,Z 734.493,A -85,B 0,C 180,E1 11738.946,E2 11738.946} C_VEL
LIN {X 0,Y 302.083,Z 715.077,A -85,B 0,C 180,E1 11736.619,E2 11736.619} C_VEL
LIN {X 0,Y 308.411,Z 698.628,A -85,B 0,C 180,E1 11735.017,E2 11735.017} C_VEL
LIN {X 0,Y 315.177,Z 678.991,A -85,B 0,C 180,E1 11733.456,E2 11733.456} C_VEL
LIN {X 0,Y 320.875,Z 659.116,A -85,B 0,C 180,E1 11732.223,E2 11732.223} C_VEL
LIN {X 0,Y 325.18,Z 641.365,A -85,B 0,C 180,E1 11731.351,E2 11731.351} C_VEL
LIN {X 0,Y 329.271,Z 620.781,A -85,B 0,C 180,E1 11730.578,E2 11730.578} C_VEL
LIN {X 0,Y 332.285,Z 598.251,A -85,B 0,C 180,E1 11729.964,E2 11729.964} C_VEL
LIN {X 0,Y 344.838,Z 432.767,A -85,B 0,C 180,E1 11726.576,E2 11726.576} C_VEL
LIN {X 0,Y 338.623,Z 420.009,A -85,B 0,C 180,E1 11723.769,E2 11723.769} C_VEL
LIN {X 0,Y 334.593,Z 412.505,A -85,B 0,C 180,E1 11721.749,E2 11721.749} C_VEL
LIN {X 0,Y 329.507,Z 404.798,A -85,B 0,C 180,E1 11718.946,E2 11718.946} C_VEL
LIN {X 0,Y 326.06,Z 399.799,A -85,B 0,C 180,E1 11716.753,E2 11716.753} C_VEL
LIN {X 0,Y 323.359,Z 395.852,A -85,B 0,C 180,E1 11714.779,E2 11714.779} C_VEL
LIN {X 0,Y 320.069,Z 391.012,A -85,B 0,C 180,E1 11711.898,E2 11711.898} C_VEL
LIN {X 0,Y 317.033,Z 387.044,A -85,B 0,C 180,E1 11708.433,E2 11708.433} C_VEL
LIN {X 0,Y 316.423,Z 385.64,A -85,B 0,C 180,E1 11707.444,E2 11707.444} C_VEL
LIN {X 0,Y 313.909,Z 383.337,A -85,B 0,C 180,E1 11700.548,E2 11700.548} C_VEL
LIN {X 0,Y 314.309,Z 383.962,A -85,B 0,C 180,E1 11696.534,E2 11696.534} C_VEL
LIN {X 0,Y 316.605,Z 385.938,A -85,B 0,C 180,E1 11691.83,E2 11691.83} C_VEL
LIN {X 0,Y 318.923,Z 389.908,A -85,B 0,C 180,E1 11688.792,E2 11688.792} C_VEL
LIN {X 0,Y 320.542,Z 391.724,A -85,B 0,C 180,E1 11687.205,E2 11687.205} C_VEL
LIN {X 0,Y 323.856,Z 396.335,A -85,B 0,C 180,E1 11684.419,E2 11684.419} C_VEL
LIN {X 0,Y 325.706,Z 398.18,A -85,B 0,C 180,E1 11683.136,E2 11683.136} C_VEL
LIN {X 0,Y 329.893,Z 402.68,A -85,B 0,C 180,E1 11680.525,E2 11680.525} C_VEL
LIN {X 0,Y 334.644,Z 406.025,A -85,B 0,C 180,E1 11677.608,E2 11677.608} C_VEL
LIN {X 0,Y 337.794,Z 409.4,A -85,B 0,C 180,E1 11675.324,E2 11675.324} C_VEL
LIN {X 0,Y 341.069,Z 411.925,A -85,B 0,C 180,E1 11672.786,E2 11672.786} C_VEL
LIN {X 0,Y 343.866,Z 413.745,A -85,B 0,C 180,E1 11670.28,E2 11670.28} C_VEL
LIN {X 0,Y 346.228,Z 417.016,A -85,B 0,C 180,E1 11667.707,E2 11667.707} C_VEL
LIN {X 0,Y 349.322,Z 419.585,A -85,B 0,C 180,E1 11664.476,E2 11664.476} C_VEL
LIN {X 0,Y 351.112,Z 420.755,A -85,B 0,C 180,E1 11662.607,E2 11662.607} C_VEL
LIN {X 0,Y 353.488,Z 424.103,A -85,B 0,C 180,E1 11659.841,E2 11659.841} C_VEL
LIN {X 0,Y 356.378,Z 426.514,A -85,B 0,C 180,E1 11656.577,E2 11656.577} C_VEL
LIN {X 0,Y 358.607,Z 427.936,A -85,B 0,C 180,E1 11654,E2 11654} C_VEL
LIN {X 0,Y 361.023,Z 431.274,A -85,B 0,C 180,E1 11650.881,E2 11650.881} C_VEL
LIN {X 0,Y 363.626,Z 433.537,A -85,B 0,C 180,E1 11647.377,E2 11647.377} C_VEL
LIN {X 0,Y 366.202,Z 434.894,A -85,B 0,C 180,E1 11643.899,E2 11643.899} C_VEL
LIN {X 0,Y 368.337,Z 438.25,A -85,B 0,C 180,E1 11640.321,E2 11640.321} C_VEL
LIN {X 0,Y 370.268,Z 440.092,A -85,B 0,C 180,E1 11636.986,E2 11636.986} C_VEL
LIN {X 0,Y 372.297,Z 441.315,A -85,B 0,C 180,E1 11633.252,E2 11633.252} C_VEL
LIN {X 0,Y 373.887,Z 442.094,A -85,B 0,C 180,E1 11629.854,E2 11629.854} C_VEL
LIN {X 0,Y 374.935,Z 443.648,A -85,B 0,C 180,E1 11627.058,E2 11627.058} C_VEL
LIN {X 0,Y 375.992,Z 445.333,A -85,B 0,C 180,E1 11623.533,E2 11623.533} C_VEL
LIN {X 0,Y 376.799,Z 446.321,A -85,B 0,C 180,E1 11620.241,E2 11620.241} C_VEL
LIN {X 0,Y 377.493,Z 446.964,A -85,B 0,C 180,E1 11616.387,E2 11616.387} C_VEL
LIN {X 0,Y 377.846,Z 447.231,A -85,B 0,C 180,E1 11613.034,E2 11613.034} C_VEL
LIN {X 0,Y 377.93,Z 447.308,A -85,B 0,C 180,E1 11609.242,E2 11609.242} C_VEL
LIN {X 0,Y 377.76,Z 447.202,A -85,B 0,C 180,E1 11605.902,E2 11605.902} C_VEL
LIN {X 0,Y 377.275,Z 446.797,A -85,B 0,C 180,E1 11602.232,E2 11602.232} C_VEL
LIN {X 0,Y 376.625,Z 446.099,A -85,B 0,C 180,E1 11598.981,E2 11598.981} C_VEL
LIN {X 0,Y 375.691,Z 444.911,A -85,B 0,C 180,E1 11595.355,E2 11595.355} C_VEL
LIN {X 0,Y 374.688,Z 443.172,A -85,B 0,C 180,E1 11592.29,E2 11592.29} C_VEL
LIN {X 0,Y 373.67,Z 441.892,A -85,B 0,C 180,E1 11589.645,E2 11589.645} C_VEL
LIN {X 0,Y 371.975,Z 441.127,A -85,B 0,C 180,E1 11586.051,E2 11586.051} C_VEL
LIN {X 0,Y 370.053,Z 439.949,A -85,B 0,C 180,E1 11582.657,E2 11582.657} C_VEL
LIN {X 0,Y 368.056,Z 437.845,A -85,B 0,C 180,E1 11579.142,E2 11579.142} C_VEL
LIN {X 0,Y 365.841,Z 434.647,A -85,B 0,C 180,E1 11575.627,E2 11575.627} C_VEL
LIN {X 0,Y 363.44,Z 433.404,A -85,B 0,C 180,E1 11572.358,E2 11572.358} C_VEL
LIN {X 0,Y 360.853,Z 431.097,A -85,B 0,C 180,E1 11568.908,E2 11568.908} C_VEL
LIN {X 0,Y 358.533,Z 427.803,A -85,B 0,C 180,E1 11565.908,E2 11565.908} C_VEL
LIN {X 0,Y 355.365,Z 425.784,A -85,B 0,C 180,E1 11562.257,E2 11562.257} C_VEL
LIN {X 0,Y 352.376,Z 422.696,A -85,B 0,C 180,E1 11558.835,E2 11558.835} C_VEL
LIN {X 0,Y 350.614,Z 420.22,A -85,B 0,C 180,E1 11556.788,E2 11556.788} C_VEL
LIN {X 0,Y 347.26,Z 417.993,A -85,B 0,C 180,E1 11553.363,E2 11553.363} C_VEL
LIN {X 0,Y 344.527,Z 414.822,A -85,B 0,C 180,E1 11550.435,E2 11550.435} C_VEL
LIN {X 0,Y 343.428,Z 413.232,A -85,B 0,C 180,E1 11549.282,E2 11549.282} C_VEL
LIN {X 0,Y 339.991,Z 411.227,A -85,B 0,C 180,E1 11546.364,E2 11546.364} C_VEL
LIN {X 0,Y 336.078,Z 407.704,A -85,B 0,C 180,E1 11543.401,E2 11543.401} C_VEL
LIN {X 0,Y 333.779,Z 405.264,A -85,B 0,C 180,E1 11541.805,E2 11541.805} C_VEL
LIN {X 0,Y 329.19,Z 402.091,A -85,B 0,C 180,E1 11539.057,E2 11539.057} C_VEL
LIN {X 0,Y 324.589,Z 396.969,A -85,B 0,C 180,E1 11536.095,E2 11536.095} C_VEL
LIN {X 0,Y 321.086,Z 392.749,A -85,B 0,C 180,E1 11533.323,E2 11533.323} C_VEL
LIN {X 0,Y 319.996,Z 390.944,A -85,B 0,C 180,E1 11532.267,E2 11532.267} C_VEL
LIN {X 0,Y 317.047,Z 387.063,A -85,B 0,C 180,E1 11528.889,E2 11528.889} C_VEL
LIN {X 0,Y 316.375,Z 385.609,A -85,B 0,C 180,E1 11527.81,E2 11527.81} C_VEL
LIN {X 0,Y 313.903,Z 383.343,A -85,B 0,C 180,E1 11520.913,E2 11520.913} C_VEL
LIN {X 0,Y 314.327,Z 383.992,A -85,B 0,C 180,E1 11516.9,E2 11516.9} C_VEL
LIN {X 0,Y 316.592,Z 385.925,A -85,B 0,C 180,E1 11512.286,E2 11512.286} C_VEL
LIN {X 0,Y 318.986,Z 389.993,A -85,B 0,C 180,E1 11509.16,E2 11509.16} C_VEL
LIN {X 0,Y 320.519,Z 391.711,A -85,B 0,C 180,E1 11507.662,E2 11507.662} C_VEL
LIN {X 0,Y 323.709,Z 396.204,A -85,B 0,C 180,E1 11504.962,E2 11504.962} C_VEL
LIN {X 0,Y 327.998,Z 402.617,A -85,B 0,C 180,E1 11501.976,E2 11501.976} C_VEL
LIN {X 0,Y 331.893,Z 408.389,A -85,B 0,C 180,E1 11499.684,E2 11499.684} C_VEL
LIN {X 0,Y 335.783,Z 414.536,A -85,B 0,C 180,E1 11497.642,E2 11497.642} C_VEL
LIN {X 0,Y 339.881,Z 422.451,A -85,B 0,C 180,E1 11495.637,E2 11495.637} C_VEL
LIN {X 0,Y 340.955,Z 426.469,A -85,B 0,C 180,E1 11495.05,E2 11495.05} C_VEL
LIN {X 0,Y 341.39,Z 432.532,A -85,B 0,C 180,E1 11494.605,E2 11494.605} C_VEL
LIN {X 0,Y 341.049,Z 440.385,A -85,B 0,C 180,E1 11494.35,E2 11494.35} C_VEL
LIN {X 0,Y 339.393,Z 457.12,A -85,B 0,C 180,E1 11494.133,E2 11494.133} C_VEL
LIN {X 0,Y 328.255,Z 599.062,A -85,B 0,C 180,E1 11491.227,E2 11491.227} C_VEL
LIN {X 0,Y 324.661,Z 623.639,A -85,B 0,C 180,E1 11490.536,E2 11490.536} C_VEL
LIN {X 0,Y 320.885,Z 641.897,A -85,B 0,C 180,E1 11489.843,E2 11489.843} C_VEL
LIN {X 0,Y 316.12,Z 660.844,A -85,B 0,C 180,E1 11488.907,E2 11488.907} C_VEL
LIN {X 0,Y 309.415,Z 682.686,A -85,B 0,C 180,E1 11487.499,E2 11487.499} C_VEL
LIN {X 0,Y 303.409,Z 699.461,A -85,B 0,C 180,E1 11486.142,E2 11486.142} C_VEL
LIN {X 0,Y 296.349,Z 717.137,A -85,B 0,C 180,E1 11484.399,E2 11484.399} C_VEL
LIN {X 0,Y 288.075,Z 735.471,A -85,B 0,C 180,E1 11482.147,E2 11482.147} C_VEL
LIN {X 0,Y 280.857,Z 750.165,A -85,B 0,C 180,E1 11479.941,E2 11479.941} C_VEL
LIN {X 0,Y 272.985,Z 765.233,A -85,B 0,C 180,E1 11477.222,E2 11477.222} C_VEL
LIN {X 0,Y 264.405,Z 780.552,A -85,B 0,C 180,E1 11473.789,E2 11473.789} C_VEL
LIN {X 0,Y 257.791,Z 792.007,A -85,B 0,C 180,E1 11470.661,E2 11470.661} C_VEL
LIN {X 0,Y 250.868,Z 803.994,A -85,B 0,C 180,E1 11466.714,E2 11466.714} C_VEL
LIN {X 0,Y 244.473,Z 815.059,A -85,B 0,C 180,E1 11462.118,E2 11462.118} C_VEL
LIN {X 0,Y 240.109,Z 823.09,A -85,B 0,C 180,E1 11458.017,E2 11458.017} C_VEL
LIN {X 0,Y 236.204,Z 831.174,A -85,B 0,C 180,E1 11452.919,E2 11452.919} C_VEL
LIN {X 0,Y 233.682,Z 837.356,A -85,B 0,C 180,E1 11447.685,E2 11447.685} C_VEL
LIN {X 0,Y 232.557,Z 841.197,A -85,B 0,C 180,E1 11443.424,E2 11443.424} C_VEL
LIN {X 0,Y 232.053,Z 844.121,A -85,B 0,C 180,E1 11438.923,E2 11438.923} C_VEL
LIN {X 0,Y 231.971,Z 846.058,A -85,B 0,C 180,E1 11433.954,E2 11433.954} C_VEL
LIN {X 0,Y 231.994,Z 846.431,A -85,B 0,C 180,E1 11429.123,E2 11429.123} C_VEL
LIN {X 0,Y 231.972,Z 845.645,A -85,B 0,C 180,E1 11424.807,E2 11424.807} C_VEL
LIN {X 0,Y 232.08,Z 843.842,A -85,B 0,C 180,E1 11420.578,E2 11420.578} C_VEL
LIN {X 0,Y 232.615,Z 840.957,A -85,B 0,C 180,E1 11416.269,E2 11416.269} C_VEL
LIN {X 0,Y 234.061,Z 836.343,A -85,B 0,C 180,E1 11411.314,E2 11411.314} C_VEL
LIN {X 0,Y 237.012,Z 829.334,A -85,B 0,C 180,E1 11405.846,E2 11405.846} C_VEL
LIN {X 0,Y 240.604,Z 822.139,A -85,B 0,C 180,E1 11401.453,E2 11401.453} C_VEL
LIN {X 0,Y 245.942,Z 812.56,A -85,B 0,C 180,E1 11396.714,E2 11396.714} C_VEL
LIN {X 0,Y 252.303,Z 801.43,A -85,B 0,C 180,E1 11392.391,E2 11392.391} C_VEL
LIN {X 0,Y 258.63,Z 790.569,A -85,B 0,C 180,E1 11388.913,E2 11388.913} C_VEL
LIN {X 0,Y 266.785,Z 776.47,A -85,B 0,C 180,E1 11385.205,E2 11385.205} C_VEL
LIN {X 0,Y 274.854,Z 761.654,A -85,B 0,C 180,E1 11382.091,E2 11382.091} C_VEL
LIN {X 0,Y 282.227,Z 747.47,A -85,B 0,C 180,E1 11379.62,E2 11379.62} C_VEL
LIN {X 0,Y 291.088,Z 729.031,A -85,B 0,C 180,E1 11377.004,E2 11377.004} C_VEL
LIN {X 0,Y 298.242,Z 712.511,A -85,B 0,C 180,E1 11375.116,E2 11375.116} C_VEL
LIN {X 0,Y 304.733,Z 695.987,A -85,B 0,C 180,E1 11373.553,E2 11373.553} C_VEL
LIN {X 0,Y 312.148,Z 674.29,A -85,B 0,C 180,E1 11371.917,E2 11371.917} C_VEL
LIN {X 0,Y 317.172,Z 656.889,A -85,B 0,C 180,E1 11370.883,E2 11370.883} C_VEL
LIN {X 0,Y 321.608,Z 638.768,A -85,B 0,C 180,E1 11370.024,E2 11370.024} C_VEL
LIN {X 0,Y 326.137,Z 614.993,A -85,B 0,C 180,E1 11369.197,E2 11369.197} C_VEL
LIN {X 0,Y 328.595,Z 595.478,A -85,B 0,C 180,E1 11368.692,E2 11368.692} C_VEL
LIN {X 0,Y 340.953,Z 436.74,A -85,B 0,C 180,E1 11365.443,E2 11365.443} C_VEL
LIN {X 0,Y 335.043,Z 424.452,A -85,B 0,C 180,E1 11362.596,E2 11362.596} C_VEL
LIN {X 0,Y 331.945,Z 418.777,A -85,B 0,C 180,E1 11360.958,E2 11360.958} C_VEL
LIN {X 0,Y 327.402,Z 411.782,A -85,B 0,C 180,E1 11358.334,E2 11358.334} C_VEL
LIN {X 0,Y 324.327,Z 407.174,A -85,B 0,C 180,E1 11356.292,E2 11356.292} C_VEL
LIN {X 0,Y 321.821,Z 403.42,A -85,B 0,C 180,E1 11354.392,E2 11354.392} C_VEL
LIN {X 0,Y 318.542,Z 398.577,A -85,B 0,C 180,E1 11351.405,E2 11351.405} C_VEL
LIN {X 0,Y 315.693,Z 394.462,A -85,B 0,C 180,E1 11347.919,E2 11347.919} C_VEL
LIN {X 0,Y 315.209,Z 393.469,A -85,B 0,C 180,E1 11347.106,E2 11347.106} C_VEL
LIN {X 0,Y 312.923,Z 391.273,A -85,B 0,C 180,E1 11340.366,E2 11340.366} C_VEL
LIN {X 0,Y 313.437,Z 392.049,A -85,B 0,C 180,E1 11336.159,E2 11336.159} C_VEL
LIN {X 0,Y 315.448,Z 393.778,A -85,B 0,C 180,E1 11332.075,E2 11332.075} C_VEL
LIN {X 0,Y 317.782,Z 397.8,A -85,B 0,C 180,E1 11328.935,E2 11328.935} C_VEL
LIN {X 0,Y 319.187,Z 399.445,A -85,B 0,C 180,E1 11327.517,E2 11327.517} C_VEL
LIN {X 0,Y 322.538,Z 404.139,A -85,B 0,C 180,E1 11324.63,E2 11324.63} C_VEL
LIN {X 0,Y 324.351,Z 406.076,A -85,B 0,C 180,E1 11323.34,E2 11323.34} C_VEL
LIN {X 0,Y 328.662,Z 410.602,A -85,B 0,C 180,E1 11320.634,E2 11320.634} C_VEL
LIN {X 0,Y 333.335,Z 413.896,A -85,B 0,C 180,E1 11317.794,E2 11317.794} C_VEL
LIN {X 0,Y 336.847,Z 417.522,A -85,B 0,C 180,E1 11315.258,E2 11315.258} C_VEL
LIN {X 0,Y 340.154,Z 419.952,A -85,B 0,C 180,E1 11312.706,E2 11312.706} C_VEL
LIN {X 0,Y 342.674,Z 421.626,A -85,B 0,C 180,E1 11310.455,E2 11310.455} C_VEL
LIN {X 0,Y 345.181,Z 424.98,A -85,B 0,C 180,E1 11307.756,E2 11307.756} C_VEL
LIN {X 0,Y 348.251,Z 427.5,A -85,B 0,C 180,E1 11304.552,E2 11304.552} C_VEL
LIN {X 0,Y 349.901,Z 428.501,A -85,B 0,C 180,E1 11302.867,E2 11302.867} C_VEL
LIN {X 0,Y 352.349,Z 431.953,A -85,B 0,C 180,E1 11300.01,E2 11300.01} C_VEL
LIN {X 0,Y 355.166,Z 434.342,A -85,B 0,C 180,E1 11296.812,E2 11296.812} C_VEL
